SPLINE
SPL {X  -157.404, Y  +360.095, Z    +0.000, E1   +17.695, E3 +134667.595}
SPL {X  -159.413, Y  +375.108, Z    +0.000, E1    +9.284, E3 +134676.684}
SPL {X  -159.978, Y  +386.135, Z    +0.000, E1    +2.544, E3 +134680.245}
SPL {X  -160.000, Y  +393.708, Z    +0.000, E1    -3.216, E3 +134681.999}
SPL {X  -160.000, Y  +400.474, Z    +0.000, E1    -9.529, E3 +134684.045}
SPL {X  -160.000, Y  +409.652, Z    +0.000, E1   -18.026, E3 +134688.182}
SPL {X  -160.000, Y  +437.804, Z    +0.000, E1   -34.779, E3 +134712.975}
SPL {X  -160.000, Y  +463.067, Z    +0.000, E1   -38.672, E3 +134758.675}
SPL {X  -160.000, Y  +469.167, Z    +0.000, E1   -38.717, E3 +134774.781}
SPL {X  -160.000, Y  +476.691, Z    +0.000, E1   -38.728, E3 +134794.712}
SPL {X  -160.000, Y  +483.419, Z    +0.000, E1   -38.692, E3 +134812.613}
SPL {X  -160.000, Y  +489.013, Z    +0.000, E1   -38.683, E3 +134827.451}
SPL {X  -160.000, Y  +494.786, Z    +0.000, E1   -38.693, E3 +134842.761}
SPL {X  -160.000, Y  +500.108, Z    +0.000, E1   -38.668, E3 +134856.913}
SPL {X  -160.000, Y  +504.903, Z    +0.000, E1   -38.673, E3 +134869.634}
SPL {X  -160.000, Y  +510.180, Z    +0.000, E1   -38.675, E3 +134883.638}
SPL {X  -160.000, Y  +515.083, Z    +0.000, E1   -38.662, E3 +134896.658}
SPL {X  -160.000, Y  +520.479, Z    +0.000, E1   -38.692, E3 +134910.932}
SPL {X  -160.000, Y  +525.998, Z    +0.000, E1   -38.666, E3 +134925.611}
SPL {X  -160.000, Y  +531.341, Z    +0.000, E1   -38.684, E3 +134939.755}
SPL {X  -160.000, Y  +537.313, Z    +0.000, E1   -38.686, E3 +134955.595}
SPL {X  -160.000, Y  +543.203, Z    +0.000, E1   -38.679, E3 +134971.220}
SPL {X  -160.000, Y  +551.201, Z    +0.000, E1   -38.768, E3 +134992.281}
SPL {X  -160.000, Y  +561.335, Z    +0.000, E1   -38.777, E3 +135019.152}
SPL {X  -160.000, Y  +568.812, Z    +0.000, E1   -38.671, E3 +135039.155}
SPL {X  -160.000, Y  +574.116, Z    +0.000, E1   -38.680, E3 +135053.225}
SPL {X  -160.000, Y  +582.193, Z    +0.000, E1   -38.759, E3 +135074.529}
SPL {X  -160.000, Y  +591.932, Z    +0.000, E1   -38.763, E3 +135100.354}
SPL {X  -160.000, Y  +601.488, Z    +0.000, E1   -38.747, E3 +135125.729}
SPL {X  -160.000, Y  +609.161, Z    +0.000, E1   -38.685, E3 +135146.181}
SPL {X  -160.000, Y  +614.445, Z    +0.000, E1   -38.661, E3 +135160.230}
SPL {X  -160.000, Y  +621.895, Z    +0.000, E1   -38.769, E3 +135179.818}
SPL {X  -160.000, Y  +631.692, Z    +0.000, E1   -38.748, E3 +135205.871}
SPL {X  -160.000, Y  +639.246, Z    +0.000, E1   -38.671, E3 +135226.047}
SPL {X  -160.000, Y  +644.827, Z    +0.000, E1   -38.662, E3 +135240.882}
SPL {X  -160.000, Y  +650.491, Z    +0.000, E1   -38.673, E3 +135255.869}
SPL {X  -160.000, Y  +656.011, Z    +0.000, E1   -38.669, E3 +135270.522}
SPL {X  -160.000, Y  +661.156, Z    +0.000, E1   -38.659, E3 +135284.197}
SPL {X  -160.000, Y  +666.701, Z    +0.000, E1   -38.683, E3 +135298.858}
SPL {X  -159.961, Y  +675.011, Z    +0.000, E1   -38.755, E3 +135320.844}
SPL {X  -159.451, Y  +684.743, Z    +0.000, E1   -38.666, E3 +135347.198}
SPL {X  -158.386, Y  +694.170, Z    +0.000, E1   -38.484, E3 +135373.316}
SPL {X  -157.286, Y  +700.846, Z    +0.000, E1   -38.194, E3 +135392.284}
SPL {X  -156.328, Y  +705.580, Z    +0.000, E1   -38.037, E3 +135405.820}
SPL {X  -155.162, Y  +710.549, Z    +0.000, E1   -37.822, E3 +135420.224}
SPL {X  -153.914, Y  +715.210, Z    +0.000, E1   -37.596, E3 +135433.873}
SPL {X  -152.686, Y  +719.322, Z    +0.000, E1   -37.361, E3 +135446.045}
SPL {X  -150.251, Y  +726.496, Z    +0.000, E1   -33.848, E3 +135494.541}
ENDSPLINE

SPLINE
SPL {X  -156.089, Y  +706.662, Z    +0.000, E1   -21.279, E3 +135547.194}
SPL {X  -159.059, Y  +688.824, Z    +0.000, E1   -11.551, E3 +135561.155}
SPL {X  -159.959, Y  +675.119, Z    +0.000, E1    -3.373, E3 +135565.983}
SPL {X  -160.000, Y  +666.447, Z    +0.000, E1    +3.005, E3 +135568.018}
SPL {X  -160.000, Y  +658.774, Z    +0.000, E1   +10.317, E3 +135570.276}
SPL {X  -160.000, Y  +647.765, Z    +0.000, E1   +20.359, E3 +135575.642}
SPL {X  -160.000, Y  +622.607, Z    +0.000, E1   +34.692, E3 +135598.509}
SPL {X  -160.000, Y  +593.120, Z    +0.000, E1   +39.775, E3 +135648.039}
SPL {X  -160.000, Y  +586.287, Z    +0.000, E1   +39.762, E3 +135665.506}
SPL {X  -160.000, Y  +577.753, Z    +0.000, E1   +39.844, E3 +135687.147}
SPL {X  -160.000, Y  +567.367, Z    +0.000, E1   +39.853, E3 +135713.642}
SPL {X  -160.000, Y  +559.466, Z    +0.000, E1   +39.761, E3 +135733.923}
SPL {X  -160.000, Y  +552.914, Z    +0.000, E1   +39.787, E3 +135750.590}
SPL {X  -160.000, Y  +546.390, Z    +0.000, E1   +39.760, E3 +135767.304}
SPL {X  -160.000, Y  +540.123, Z    +0.000, E1   +39.770, E3 +135783.283}
SPL {X  -160.000, Y  +533.658, Z    +0.000, E1   +39.771, E3 +135799.782}
SPL {X  -160.000, Y  +527.046, Z    +0.000, E1   +39.771, E3 +135816.658}
SPL {X  -160.000, Y  +521.063, Z    +0.000, E1   +39.756, E3 +135831.942}
SPL {X  -160.000, Y  +515.110, Z    +0.000, E1   +39.770, E3 +135847.115}
SPL {X  -160.000, Y  +508.717, Z    +0.000, E1   +39.766, E3 +135863.433}
SPL {X  -160.000, Y  +502.133, Z    +0.000, E1   +39.780, E3 +135880.199}
ENDSPLINE

SPLINE
SPL {X  -160.000, Y  +512.949, Z    +0.000, E1   +32.050, E3 +135896.457}
ENDSPLINE

SPLINE
SPL {X  -160.000, Y  +507.092, Z    +0.000, E1   +32.805, E3 +135911.085}
SPL {X  -160.000, Y  +499.824, Z    +0.000, E1   +34.003, E3 +135926.827}
SPL {X  -160.000, Y  +491.367, Z    +0.000, E1   +35.449, E3 +135943.568}
SPL {X  -160.000, Y  +483.082, Z    +0.000, E1   +36.782, E3 +135959.406}
SPL {X  -160.000, Y  +474.521, Z    +0.000, E1   +38.037, E3 +135975.494}
SPL {X  -160.000, Y  +465.343, Z    +0.000, E1   +38.802, E3 +135995.653}
SPL {X  -160.000, Y  +457.266, Z    +0.000, E1   +38.756, E3 +136017.107}
SPL {X  -160.000, Y  +448.553, Z    +0.000, E1   +38.823, E3 +136040.058}
SPL {X  -160.000, Y  +439.425, Z    +0.000, E1   +38.797, E3 +136064.229}
SPL {X  -160.000, Y  +430.351, Z    +0.000, E1   +38.810, E3 +136088.244}
SPL {X  -160.000, Y  +421.477, Z    +0.000, E1   +38.792, E3 +136111.747}
SPL {X  -160.000, Y  +412.292, Z    +0.000, E1   +38.825, E3 +136135.975}
SPL {X  -160.000, Y  +403.281, Z    +0.000, E1   +38.797, E3 +136159.855}
SPL {X  -160.000, Y  +394.948, Z    +0.000, E1   +38.796, E3 +136181.896}
SPL {X  -159.971, Y  +385.741, Z    +0.000, E1   +38.831, E3 +136206.218}
SPL {X  -159.525, Y  +376.478, Z    +0.000, E1   +38.739, E3 +136231.209}
SPL {X  -158.721, Y  +368.613, Z    +0.000, E1   +38.561, E3 +136252.932}
SPL {X  -157.505, Y  +360.654, Z    +0.000, E1   +38.390, E3 +136275.205}
SPL {X  -156.229, Y  +354.269, Z    +0.000, E1   +38.076, E3 +136293.555}
SPL {X  -155.202, Y  +349.910, Z    +0.000, E1   +37.893, E3 +136306.129}
SPL {X  -154.128, Y  +345.852, Z    +0.000, E1   +37.701, E3 +136317.953}
SPL {X  -152.890, Y  +341.633, Z    +0.000, E1   +37.487, E3 +136330.385}
SPL {X  -150.284, Y  +333.893, Z    +0.000, E1   +33.433, E3 +136385.195}
ENDSPLINE

SPLINE
SPL {X  -157.404, Y  +360.095, Z    +0.000, E1   +17.695, E3 +136440.320}
SPL {X  -159.413, Y  +375.108, Z    +0.000, E1    +9.284, E3 +136449.409}
SPL {X  -159.978, Y  +386.135, Z    +0.000, E1    +2.544, E3 +136452.970}
SPL {X  -160.000, Y  +393.708, Z    +0.000, E1    -3.216, E3 +136454.724}
SPL {X  -160.000, Y  +400.474, Z    +0.000, E1    -9.529, E3 +136456.771}
SPL {X  -160.000, Y  +409.652, Z    +0.000, E1   -18.026, E3 +136460.907}
SPL {X  -160.000, Y  +437.804, Z    +0.000, E1   -34.779, E3 +136485.700}
SPL {X  -160.000, Y  +463.067, Z    +0.000, E1   -38.672, E3 +136531.400}
SPL {X  -160.000, Y  +469.167, Z    +0.000, E1   -38.717, E3 +136547.506}
SPL {X  -160.000, Y  +476.691, Z    +0.000, E1   -38.728, E3 +136567.438}
SPL {X  -160.000, Y  +483.419, Z    +0.000, E1   -38.692, E3 +136585.338}
SPL {X  -160.000, Y  +489.013, Z    +0.000, E1   -38.683, E3 +136600.177}
SPL {X  -160.000, Y  +494.786, Z    +0.000, E1   -38.693, E3 +136615.487}
SPL {X  -160.000, Y  +500.108, Z    +0.000, E1   -38.668, E3 +136629.638}
SPL {X  -160.000, Y  +504.903, Z    +0.000, E1   -38.673, E3 +136642.359}
SPL {X  -160.000, Y  +510.180, Z    +0.000, E1   -38.675, E3 +136656.363}
SPL {X  -160.000, Y  +515.083, Z    +0.000, E1   -38.662, E3 +136669.383}
SPL {X  -160.000, Y  +520.479, Z    +0.000, E1   -38.692, E3 +136683.658}
SPL {X  -160.000, Y  +525.998, Z    +0.000, E1   -38.666, E3 +136698.336}
SPL {X  -160.000, Y  +531.341, Z    +0.000, E1   -38.684, E3 +136712.480}
SPL {X  -160.000, Y  +537.313, Z    +0.000, E1   -38.686, E3 +136728.320}
SPL {X  -160.000, Y  +543.203, Z    +0.000, E1   -38.679, E3 +136743.945}
SPL {X  -160.000, Y  +551.201, Z    +0.000, E1   -38.768, E3 +136765.007}
SPL {X  -160.000, Y  +561.335, Z    +0.000, E1   -38.777, E3 +136791.877}
SPL {X  -160.000, Y  +568.812, Z    +0.000, E1   -38.671, E3 +136811.880}
SPL {X  -160.000, Y  +574.116, Z    +0.000, E1   -38.680, E3 +136825.951}
SPL {X  -160.000, Y  +582.193, Z    +0.000, E1   -38.759, E3 +136847.254}
SPL {X  -160.000, Y  +591.932, Z    +0.000, E1   -38.763, E3 +136873.079}
SPL {X  -160.000, Y  +601.488, Z    +0.000, E1   -38.747, E3 +136898.454}
SPL {X  -160.000, Y  +609.161, Z    +0.000, E1   -38.685, E3 +136918.906}
SPL {X  -160.000, Y  +614.445, Z    +0.000, E1   -38.661, E3 +136932.955}
SPL {X  -160.000, Y  +621.895, Z    +0.000, E1   -38.769, E3 +136952.543}
SPL {X  -160.000, Y  +631.692, Z    +0.000, E1   -38.748, E3 +136978.597}
SPL {X  -160.000, Y  +639.246, Z    +0.000, E1   -38.671, E3 +136998.772}
SPL {X  -160.000, Y  +644.827, Z    +0.000, E1   -38.662, E3 +137013.607}
SPL {X  -160.000, Y  +650.491, Z    +0.000, E1   -38.673, E3 +137028.595}
SPL {X  -160.000, Y  +656.011, Z    +0.000, E1   -38.669, E3 +137043.248}
SPL {X  -160.000, Y  +661.156, Z    +0.000, E1   -38.659, E3 +137056.923}
SPL {X  -160.000, Y  +666.701, Z    +0.000, E1   -38.683, E3 +137071.583}
SPL {X  -159.961, Y  +675.011, Z    +0.000, E1   -38.755, E3 +137093.569}
SPL {X  -159.451, Y  +684.743, Z    +0.000, E1   -38.666, E3 +137119.923}
SPL {X  -158.386, Y  +694.170, Z    +0.000, E1   -38.484, E3 +137146.041}
SPL {X  -157.286, Y  +700.846, Z    +0.000, E1   -38.194, E3 +137165.009}
SPL {X  -156.328, Y  +705.580, Z    +0.000, E1   -38.037, E3 +137178.545}
SPL {X  -155.162, Y  +710.549, Z    +0.000, E1   -37.822, E3 +137192.949}
SPL {X  -153.914, Y  +715.210, Z    +0.000, E1   -37.596, E3 +137206.598}
SPL {X  -152.686, Y  +719.322, Z    +0.000, E1   -37.361, E3 +137218.771}
SPL {X  -150.251, Y  +726.496, Z    +0.000, E1   -33.848, E3 +137267.266}
ENDSPLINE

SPLINE
SPL {X  -156.089, Y  +706.662, Z    +0.000, E1   -21.279, E3 +137319.920}
SPL {X  -159.059, Y  +688.824, Z    +0.000, E1   -11.551, E3 +137333.880}
SPL {X  -159.959, Y  +675.119, Z    +0.000, E1    -3.373, E3 +137338.708}
SPL {X  -160.000, Y  +666.447, Z    +0.000, E1    +3.005, E3 +137340.743}
SPL {X  -160.000, Y  +658.774, Z    +0.000, E1   +10.317, E3 +137343.002}
SPL {X  -160.000, Y  +647.765, Z    +0.000, E1   +20.359, E3 +137348.367}
SPL {X  -160.000, Y  +622.607, Z    +0.000, E1   +34.692, E3 +137371.234}
SPL {X  -160.000, Y  +596.106, Z    +0.000, E1   +39.718, E3 +137413.234}
SPL {X  -160.000, Y  +592.273, Z    +0.000, E1   +39.746, E3 +137422.972}
SPL {X  -160.000, Y  +586.287, Z    +0.000, E1   +39.762, E3 +137438.231}
SPL {X  -160.000, Y  +577.753, Z    +0.000, E1   +39.844, E3 +137459.873}
SPL {X  -160.000, Y  +567.367, Z    +0.000, E1   +39.853, E3 +137486.367}
SPL {X  -160.000, Y  +559.466, Z    +0.000, E1   +39.761, E3 +137506.648}
SPL {X  -160.000, Y  +552.914, Z    +0.000, E1   +39.787, E3 +137523.316}
SPL {X  -160.000, Y  +546.390, Z    +0.000, E1   +39.760, E3 +137540.029}
SPL {X  -160.000, Y  +540.123, Z    +0.000, E1   +39.770, E3 +137556.009}
SPL {X  -160.000, Y  +533.658, Z    +0.000, E1   +39.771, E3 +137572.507}
SPL {X  -160.000, Y  +527.046, Z    +0.000, E1   +39.771, E3 +137589.383}
SPL {X  -160.000, Y  +521.063, Z    +0.000, E1   +39.756, E3 +137604.667}
SPL {X  -160.000, Y  +515.110, Z    +0.000, E1   +39.770, E3 +137619.840}
SPL {X  -160.000, Y  +508.717, Z    +0.000, E1   +39.766, E3 +137636.158}
SPL {X  -160.000, Y  +502.133, Z    +0.000, E1   +39.780, E3 +137652.925}
ENDSPLINE

SPLINE
SPL {X  -160.000, Y  +512.949, Z    +0.000, E1   +32.050, E3 +137669.182}
ENDSPLINE

SPLINE
SPL {X  -160.000, Y  +507.092, Z    +0.000, E1   +32.805, E3 +137683.810}
SPL {X  -160.000, Y  +499.824, Z    +0.000, E1   +34.003, E3 +137699.552}
SPL {X  -160.000, Y  +491.367, Z    +0.000, E1   +35.449, E3 +137716.293}
SPL {X  -160.000, Y  +483.082, Z    +0.000, E1   +36.782, E3 +137732.132}
SPL {X  -160.000, Y  +474.521, Z    +0.000, E1   +38.037, E3 +137748.220}
SPL {X  -160.000, Y  +465.343, Z    +0.000, E1   +38.802, E3 +137768.378}
SPL {X  -160.000, Y  +457.266, Z    +0.000, E1   +38.756, E3 +137789.832}
SPL {X  -160.000, Y  +448.553, Z    +0.000, E1   +38.823, E3 +137812.783}
SPL {X  -160.000, Y  +439.425, Z    +0.000, E1   +38.797, E3 +137836.954}
SPL {X  -160.000, Y  +430.351, Z    +0.000, E1   +38.810, E3 +137860.969}
SPL {X  -160.000, Y  +421.477, Z    +0.000, E1   +38.792, E3 +137884.472}
SPL {X  -160.000, Y  +412.292, Z    +0.000, E1   +38.825, E3 +137908.700}
SPL {X  -160.000, Y  +403.281, Z    +0.000, E1   +38.797, E3 +137932.580}
SPL {X  -160.000, Y  +394.948, Z    +0.000, E1   +38.796, E3 +137954.621}
SPL {X  -159.971, Y  +385.741, Z    +0.000, E1   +38.831, E3 +137978.943}
SPL {X  -159.525, Y  +376.478, Z    +0.000, E1   +38.739, E3 +138003.934}
SPL {X  -158.721, Y  +368.613, Z    +0.000, E1   +38.561, E3 +138025.657}
SPL {X  -157.505, Y  +360.654, Z    +0.000, E1   +38.390, E3 +138047.930}
SPL {X  -156.229, Y  +354.269, Z    +0.000, E1   +38.076, E3 +138066.280}
SPL {X  -155.202, Y  +349.910, Z    +0.000, E1   +37.893, E3 +138078.854}
SPL {X  -154.128, Y  +345.852, Z    +0.000, E1   +37.701, E3 +138090.678}
SPL {X  -152.890, Y  +341.633, Z    +0.000, E1   +37.487, E3 +138103.110}
SPL {X  -150.284, Y  +333.893, Z    +0.000, E1   +33.433, E3 +138157.921}
ENDSPLINE

SPLINE
SPL {X  -157.404, Y  +360.095, Z    +0.000, E1   +17.695, E3 +138213.045}
SPL {X  -159.413, Y  +375.108, Z    +0.000, E1    +9.284, E3 +138222.134}
SPL {X  -159.978, Y  +386.135, Z    +0.000, E1    +2.544, E3 +138225.695}
SPL {X  -160.000, Y  +393.708, Z    +0.000, E1    -3.216, E3 +138227.449}
SPL {X  -160.000, Y  +400.474, Z    +0.000, E1    -9.529, E3 +138229.496}
SPL {X  -160.000, Y  +409.652, Z    +0.000, E1   -18.026, E3 +138233.632}
SPL {X  -160.000, Y  +437.804, Z    +0.000, E1   -34.779, E3 +138258.425}
SPL {X  -160.000, Y  +463.067, Z    +0.000, E1   -38.672, E3 +138304.125}
SPL {X  -160.000, Y  +469.167, Z    +0.000, E1   -38.717, E3 +138320.231}
SPL {X  -160.000, Y  +476.691, Z    +0.000, E1   -38.728, E3 +138340.163}
SPL {X  -160.000, Y  +483.419, Z    +0.000, E1   -38.692, E3 +138358.063}
SPL {X  -160.000, Y  +489.013, Z    +0.000, E1   -38.683, E3 +138372.902}
SPL {X  -160.000, Y  +494.786, Z    +0.000, E1   -38.693, E3 +138388.212}
SPL {X  -160.000, Y  +500.108, Z    +0.000, E1   -38.668, E3 +138402.363}
SPL {X  -160.000, Y  +504.903, Z    +0.000, E1   -38.673, E3 +138415.084}
SPL {X  -160.000, Y  +510.180, Z    +0.000, E1   -38.675, E3 +138429.089}
SPL {X  -160.000, Y  +515.083, Z    +0.000, E1   -38.662, E3 +138442.108}
SPL {X  -160.000, Y  +520.479, Z    +0.000, E1   -38.692, E3 +138456.383}
SPL {X  -160.000, Y  +525.998, Z    +0.000, E1   -38.666, E3 +138471.061}
SPL {X  -160.000, Y  +531.341, Z    +0.000, E1   -38.684, E3 +138485.205}
SPL {X  -160.000, Y  +537.313, Z    +0.000, E1   -38.686, E3 +138501.045}
SPL {X  -160.000, Y  +543.203, Z    +0.000, E1   -38.679, E3 +138516.671}
SPL {X  -160.000, Y  +551.201, Z    +0.000, E1   -38.768, E3 +138537.732}
SPL {X  -160.000, Y  +561.335, Z    +0.000, E1   -38.777, E3 +138564.602}
SPL {X  -160.000, Y  +568.812, Z    +0.000, E1   -38.671, E3 +138584.605}
SPL {X  -160.000, Y  +574.116, Z    +0.000, E1   -38.680, E3 +138598.676}
SPL {X  -160.000, Y  +582.193, Z    +0.000, E1   -38.759, E3 +138619.979}
SPL {X  -160.000, Y  +591.932, Z    +0.000, E1   -38.763, E3 +138645.804}
SPL {X  -160.000, Y  +601.488, Z    +0.000, E1   -38.747, E3 +138671.179}
SPL {X  -160.000, Y  +609.161, Z    +0.000, E1   -38.685, E3 +138691.631}
SPL {X  -160.000, Y  +614.445, Z    +0.000, E1   -38.661, E3 +138705.680}
SPL {X  -160.000, Y  +621.895, Z    +0.000, E1   -38.769, E3 +138725.269}
SPL {X  -160.000, Y  +631.692, Z    +0.000, E1   -38.748, E3 +138751.322}
SPL {X  -160.000, Y  +639.246, Z    +0.000, E1   -38.671, E3 +138771.498}
SPL {X  -160.000, Y  +644.827, Z    +0.000, E1   -38.662, E3 +138786.332}
SPL {X  -160.000, Y  +650.491, Z    +0.000, E1   -38.673, E3 +138801.320}
SPL {X  -160.000, Y  +656.011, Z    +0.000, E1   -38.669, E3 +138815.973}
SPL {X  -160.000, Y  +661.156, Z    +0.000, E1   -38.659, E3 +138829.648}
SPL {X  -160.000, Y  +666.701, Z    +0.000, E1   -38.683, E3 +138844.308}
SPL {X  -159.961, Y  +675.011, Z    +0.000, E1   -38.755, E3 +138866.295}
SPL {X  -159.451, Y  +684.743, Z    +0.000, E1   -38.666, E3 +138892.648}
SPL {X  -158.386, Y  +694.170, Z    +0.000, E1   -38.484, E3 +138918.767}
SPL {X  -157.286, Y  +700.846, Z    +0.000, E1   -38.194, E3 +138937.734}
SPL {X  -156.328, Y  +705.580, Z    +0.000, E1   -38.037, E3 +138951.270}
SPL {X  -155.162, Y  +710.549, Z    +0.000, E1   -37.822, E3 +138965.674}
SPL {X  -153.914, Y  +715.210, Z    +0.000, E1   -37.596, E3 +138979.324}
SPL {X  -152.686, Y  +719.322, Z    +0.000, E1   -37.361, E3 +138991.496}
SPL {X  -150.251, Y  +726.496, Z    +0.000, E1   -33.848, E3 +139039.992}
ENDSPLINE

SPLINE
SPL {X  -156.089, Y  +706.662, Z    +0.000, E1   -21.279, E3 +139092.645}
SPL {X  -159.059, Y  +688.824, Z    +0.000, E1   -11.551, E3 +139106.605}
SPL {X  -159.959, Y  +675.119, Z    +0.000, E1    -3.373, E3 +139111.433}
SPL {X  -160.000, Y  +666.447, Z    +0.000, E1    +3.005, E3 +139113.468}
SPL {X  -160.000, Y  +658.774, Z    +0.000, E1   +10.317, E3 +139115.727}
SPL {X  -160.000, Y  +647.765, Z    +0.000, E1   +20.359, E3 +139121.092}
SPL {X  -160.000, Y  +622.607, Z    +0.000, E1   +34.692, E3 +139143.959}
SPL {X  -160.000, Y  +596.106, Z    +0.000, E1   +39.718, E3 +139185.959}
SPL {X  -160.000, Y  +592.273, Z    +0.000, E1   +39.746, E3 +139195.697}
SPL {X  -160.000, Y  +586.287, Z    +0.000, E1   +39.762, E3 +139210.956}
SPL {X  -160.000, Y  +577.753, Z    +0.000, E1   +39.844, E3 +139232.598}
SPL {X  -160.000, Y  +567.367, Z    +0.000, E1   +39.853, E3 +139259.092}
SPL {X  -160.000, Y  +559.466, Z    +0.000, E1   +39.761, E3 +139279.373}
SPL {X  -160.000, Y  +552.914, Z    +0.000, E1   +39.787, E3 +139296.041}
SPL {X  -160.000, Y  +546.390, Z    +0.000, E1   +39.760, E3 +139312.755}
SPL {X  -160.000, Y  +540.123, Z    +0.000, E1   +39.770, E3 +139328.734}
SPL {X  -160.000, Y  +533.658, Z    +0.000, E1   +39.771, E3 +139345.232}
SPL {X  -160.000, Y  +527.046, Z    +0.000, E1   +39.771, E3 +139362.108}
SPL {X  -160.000, Y  +521.063, Z    +0.000, E1   +39.756, E3 +139377.393}
SPL {X  -160.000, Y  +515.110, Z    +0.000, E1   +39.770, E3 +139392.565}
SPL {X  -160.000, Y  +508.717, Z    +0.000, E1   +39.766, E3 +139408.884}
SPL {X  -160.000, Y  +502.133, Z    +0.000, E1   +39.780, E3 +139425.650}
ENDSPLINE

SPLINE
SPL {X  -160.000, Y  +512.949, Z    +0.000, E1   +32.050, E3 +139441.907}
ENDSPLINE

SPLINE
SPL {X  -160.000, Y  +507.092, Z    +0.000, E1   +32.805, E3 +139456.536}
SPL {X  -160.000, Y  +499.824, Z    +0.000, E1   +34.003, E3 +139472.277}
SPL {X  -160.000, Y  +491.367, Z    +0.000, E1   +35.449, E3 +139489.018}
SPL {X  -160.000, Y  +483.082, Z    +0.000, E1   +36.782, E3 +139504.857}
SPL {X  -160.000, Y  +474.521, Z    +0.000, E1   +38.037, E3 +139520.945}
SPL {X  -160.000, Y  +465.343, Z    +0.000, E1   +38.802, E3 +139541.104}
SPL {X  -160.000, Y  +457.266, Z    +0.000, E1   +38.756, E3 +139562.557}
SPL {X  -160.000, Y  +448.553, Z    +0.000, E1   +38.823, E3 +139585.508}
SPL {X  -160.000, Y  +439.425, Z    +0.000, E1   +38.797, E3 +139609.679}
SPL {X  -160.000, Y  +430.351, Z    +0.000, E1   +38.810, E3 +139633.694}
SPL {X  -160.000, Y  +421.477, Z    +0.000, E1   +38.792, E3 +139657.198}
SPL {X  -160.000, Y  +412.292, Z    +0.000, E1   +38.825, E3 +139681.425}
SPL {X  -160.000, Y  +403.281, Z    +0.000, E1   +38.797, E3 +139705.305}
SPL {X  -160.000, Y  +394.948, Z    +0.000, E1   +38.796, E3 +139727.347}
SPL {X  -159.971, Y  +385.741, Z    +0.000, E1   +38.831, E3 +139751.668}
SPL {X  -159.525, Y  +376.478, Z    +0.000, E1   +38.739, E3 +139776.659}
SPL {X  -158.721, Y  +368.613, Z    +0.000, E1   +38.561, E3 +139798.382}
SPL {X  -157.505, Y  +360.654, Z    +0.000, E1   +38.390, E3 +139820.655}
SPL {X  -156.229, Y  +354.269, Z    +0.000, E1   +38.076, E3 +139839.005}
SPL {X  -155.202, Y  +349.910, Z    +0.000, E1   +37.893, E3 +139851.580}
SPL {X  -154.128, Y  +345.852, Z    +0.000, E1   +37.701, E3 +139863.404}
SPL {X  -152.890, Y  +341.633, Z    +0.000, E1   +37.487, E3 +139875.836}
SPL {X  -150.284, Y  +333.893, Z    +0.000, E1   +33.433, E3 +139930.646}
ENDSPLINE

SPLINE
SPL {X  -157.404, Y  +360.095, Z    +0.000, E1   +17.695, E3 +139985.771}
SPL {X  -159.413, Y  +375.108, Z    +0.000, E1    +9.284, E3 +139994.860}
SPL {X  -159.978, Y  +386.135, Z    +0.000, E1    +2.544, E3 +139998.421}
SPL {X  -160.000, Y  +393.708, Z    +0.000, E1    -3.216, E3 +140000.175}
SPL {X  -160.000, Y  +400.474, Z    +0.000, E1    -9.529, E3 +140002.221}
SPL {X  -160.000, Y  +409.652, Z    +0.000, E1   -18.026, E3 +140006.358}
SPL {X  -160.000, Y  +437.804, Z    +0.000, E1   -34.779, E3 +140031.150}
SPL {X  -160.000, Y  +463.067, Z    +0.000, E1   -38.672, E3 +140076.850}
SPL {X  -160.000, Y  +469.167, Z    +0.000, E1   -38.717, E3 +140092.956}
SPL {X  -160.000, Y  +476.691, Z    +0.000, E1   -38.728, E3 +140112.888}
SPL {X  -160.000, Y  +483.419, Z    +0.000, E1   -38.692, E3 +140130.788}
SPL {X  -160.000, Y  +489.013, Z    +0.000, E1   -38.683, E3 +140145.627}
SPL {X  -160.000, Y  +494.786, Z    +0.000, E1   -38.693, E3 +140160.937}
SPL {X  -160.000, Y  +500.108, Z    +0.000, E1   -38.668, E3 +140175.089}
SPL {X  -160.000, Y  +504.903, Z    +0.000, E1   -38.673, E3 +140187.810}
SPL {X  -160.000, Y  +510.180, Z    +0.000, E1   -38.675, E3 +140201.814}
SPL {X  -160.000, Y  +515.083, Z    +0.000, E1   -38.662, E3 +140214.834}
SPL {X  -160.000, Y  +520.479, Z    +0.000, E1   -38.692, E3 +140229.108}
SPL {X  -160.000, Y  +525.998, Z    +0.000, E1   -38.666, E3 +140243.786}
SPL {X  -160.000, Y  +531.341, Z    +0.000, E1   -38.684, E3 +140257.930}
SPL {X  -160.000, Y  +537.313, Z    +0.000, E1   -38.686, E3 +140273.770}
SPL {X  -160.000, Y  +543.203, Z    +0.000, E1   -38.679, E3 +140289.396}
SPL {X  -160.000, Y  +551.201, Z    +0.000, E1   -38.768, E3 +140310.457}
SPL {X  -160.000, Y  +561.335, Z    +0.000, E1   -38.777, E3 +140337.327}
SPL {X  -160.000, Y  +568.812, Z    +0.000, E1   -38.671, E3 +140357.331}
SPL {X  -160.000, Y  +574.116, Z    +0.000, E1   -38.680, E3 +140371.401}
SPL {X  -160.000, Y  +582.193, Z    +0.000, E1   -38.759, E3 +140392.705}
SPL {X  -160.000, Y  +591.932, Z    +0.000, E1   -38.763, E3 +140418.530}
SPL {X  -160.000, Y  +601.488, Z    +0.000, E1   -38.747, E3 +140443.905}
SPL {X  -160.000, Y  +609.161, Z    +0.000, E1   -38.685, E3 +140464.357}
SPL {X  -160.000, Y  +614.445, Z    +0.000, E1   -38.661, E3 +140478.406}
SPL {X  -160.000, Y  +621.895, Z    +0.000, E1   -38.769, E3 +140497.994}
SPL {X  -160.000, Y  +631.692, Z    +0.000, E1   -38.748, E3 +140524.047}
SPL {X  -160.000, Y  +639.246, Z    +0.000, E1   -38.671, E3 +140544.223}
SPL {X  -160.000, Y  +644.827, Z    +0.000, E1   -38.662, E3 +140559.058}
SPL {X  -160.000, Y  +650.491, Z    +0.000, E1   -38.673, E3 +140574.045}
SPL {X  -160.000, Y  +656.011, Z    +0.000, E1   -38.669, E3 +140588.698}
SPL {X  -160.000, Y  +661.156, Z    +0.000, E1   -38.659, E3 +140602.373}
SPL {X  -160.000, Y  +666.701, Z    +0.000, E1   -38.683, E3 +140617.033}
SPL {X  -159.961, Y  +675.011, Z    +0.000, E1   -38.755, E3 +140639.020}
SPL {X  -159.451, Y  +684.743, Z    +0.000, E1   -38.666, E3 +140665.373}
SPL {X  -158.386, Y  +694.170, Z    +0.000, E1   -38.484, E3 +140691.492}
SPL {X  -157.286, Y  +700.846, Z    +0.000, E1   -38.194, E3 +140710.460}
SPL {X  -156.328, Y  +705.580, Z    +0.000, E1   -38.037, E3 +140723.996}
SPL {X  -155.162, Y  +710.549, Z    +0.000, E1   -37.822, E3 +140738.399}
SPL {X  -153.914, Y  +715.210, Z    +0.000, E1   -37.596, E3 +140752.049}
SPL {X  -152.686, Y  +719.322, Z    +0.000, E1   -37.361, E3 +140764.221}
SPL {X  -150.251, Y  +726.496, Z    +0.000, E1   -33.848, E3 +140812.717}
ENDSPLINE

SPLINE
SPL {X  -156.089, Y  +706.662, Z    +0.000, E1   -21.279, E3 +140865.370}
SPL {X  -159.059, Y  +688.824, Z    +0.000, E1   -11.551, E3 +140879.331}
SPL {X  -159.959, Y  +675.119, Z    +0.000, E1    -3.373, E3 +140884.159}
SPL {X  -160.000, Y  +666.447, Z    +0.000, E1    +3.005, E3 +140886.194}
SPL {X  -160.000, Y  +658.774, Z    +0.000, E1   +10.317, E3 +140888.452}
SPL {X  -160.000, Y  +647.765, Z    +0.000, E1   +20.359, E3 +140893.817}
SPL {X  -160.000, Y  +622.607, Z    +0.000, E1   +34.692, E3 +140916.685}
SPL {X  -160.000, Y  +593.120, Z    +0.000, E1   +39.775, E3 +140966.215}
SPL {X  -160.000, Y  +586.287, Z    +0.000, E1   +39.762, E3 +140983.681}
SPL {X  -160.000, Y  +577.753, Z    +0.000, E1   +39.844, E3 +141005.323}
SPL {X  -160.000, Y  +567.367, Z    +0.000, E1   +39.853, E3 +141031.817}
SPL {X  -160.000, Y  +559.466, Z    +0.000, E1   +39.761, E3 +141052.099}
SPL {X  -160.000, Y  +552.914, Z    +0.000, E1   +39.787, E3 +141068.766}
SPL {X  -160.000, Y  +546.390, Z    +0.000, E1   +39.760, E3 +141085.480}
SPL {X  -160.000, Y  +540.123, Z    +0.000, E1   +39.770, E3 +141101.459}
SPL {X  -160.000, Y  +533.658, Z    +0.000, E1   +39.771, E3 +141117.958}
SPL {X  -160.000, Y  +527.046, Z    +0.000, E1   +39.771, E3 +141134.833}
SPL {X  -160.000, Y  +521.063, Z    +0.000, E1   +39.756, E3 +141150.118}
SPL {X  -160.000, Y  +515.110, Z    +0.000, E1   +39.770, E3 +141165.290}
SPL {X  -160.000, Y  +508.717, Z    +0.000, E1   +39.766, E3 +141181.609}
SPL {X  -160.000, Y  +502.133, Z    +0.000, E1   +39.780, E3 +141198.375}
ENDSPLINE

SPLINE
SPL {X  -160.000, Y  +512.949, Z    +0.000, E1   +32.050, E3 +141214.633}
ENDSPLINE

SPLINE
SPL {X  -160.000, Y  +507.092, Z    +0.000, E1   +32.805, E3 +141229.261}
SPL {X  -160.000, Y  +499.824, Z    +0.000, E1   +34.003, E3 +141245.003}
SPL {X  -160.000, Y  +491.367, Z    +0.000, E1   +35.449, E3 +141261.743}
SPL {X  -160.000, Y  +483.082, Z    +0.000, E1   +36.782, E3 +141277.582}
SPL {X  -160.000, Y  +474.521, Z    +0.000, E1   +38.037, E3 +141293.670}
SPL {X  -160.000, Y  +465.343, Z    +0.000, E1   +38.802, E3 +141313.829}
SPL {X  -160.000, Y  +457.266, Z    +0.000, E1   +38.756, E3 +141335.283}
SPL {X  -160.000, Y  +448.553, Z    +0.000, E1   +38.823, E3 +141358.234}
SPL {X  -160.000, Y  +439.425, Z    +0.000, E1   +38.797, E3 +141382.405}
SPL {X  -160.000, Y  +430.351, Z    +0.000, E1   +38.810, E3 +141406.419}
SPL {X  -160.000, Y  +421.477, Z    +0.000, E1   +38.792, E3 +141429.923}
SPL {X  -160.000, Y  +412.292, Z    +0.000, E1   +38.825, E3 +141454.150}
SPL {X  -160.000, Y  +403.281, Z    +0.000, E1   +38.797, E3 +141478.030}
SPL {X  -160.000, Y  +394.948, Z    +0.000, E1   +38.796, E3 +141500.072}
SPL {X  -159.971, Y  +385.741, Z    +0.000, E1   +38.831, E3 +141524.393}
SPL {X  -159.525, Y  +376.478, Z    +0.000, E1   +38.739, E3 +141549.384}
SPL {X  -158.721, Y  +368.613, Z    +0.000, E1   +38.561, E3 +141571.107}
SPL {X  -157.505, Y  +360.654, Z    +0.000, E1   +38.390, E3 +141593.381}
SPL {X  -156.229, Y  +354.269, Z    +0.000, E1   +38.076, E3 +141611.730}
SPL {X  -155.202, Y  +349.910, Z    +0.000, E1   +37.893, E3 +141624.305}
SPL {X  -154.128, Y  +345.852, Z    +0.000, E1   +37.701, E3 +141636.129}
SPL {X  -152.890, Y  +341.633, Z    +0.000, E1   +37.487, E3 +141648.561}
SPL {X  -150.284, Y  +333.893, Z    +0.000, E1   +33.433, E3 +141703.371}
ENDSPLINE

SPLINE
SPL {X  -157.404, Y  +360.095, Z    +0.000, E1   +17.695, E3 +141758.496}
SPL {X  -159.413, Y  +375.108, Z    +0.000, E1    +9.284, E3 +141767.585}
SPL {X  -159.978, Y  +386.135, Z    +0.000, E1    +2.544, E3 +141771.146}
SPL {X  -160.000, Y  +393.708, Z    +0.000, E1    -3.216, E3 +141772.900}
SPL {X  -160.000, Y  +400.474, Z    +0.000, E1    -9.529, E3 +141774.946}
SPL {X  -160.000, Y  +409.652, Z    +0.000, E1   -18.026, E3 +141779.083}
SPL {X  -160.000, Y  +437.804, Z    +0.000, E1   -34.779, E3 +141803.876}
SPL {X  -160.000, Y  +463.067, Z    +0.000, E1   -38.672, E3 +141849.576}
SPL {X  -160.000, Y  +469.167, Z    +0.000, E1   -38.717, E3 +141865.682}
SPL {X  -160.000, Y  +476.691, Z    +0.000, E1   -38.728, E3 +141885.613}
SPL {X  -160.000, Y  +483.419, Z    +0.000, E1   -38.692, E3 +141903.514}
SPL {X  -160.000, Y  +489.013, Z    +0.000, E1   -38.683, E3 +141918.352}
SPL {X  -160.000, Y  +494.786, Z    +0.000, E1   -38.693, E3 +141933.662}
SPL {X  -160.000, Y  +500.108, Z    +0.000, E1   -38.668, E3 +141947.814}
SPL {X  -160.000, Y  +504.903, Z    +0.000, E1   -38.673, E3 +141960.535}
SPL {X  -160.000, Y  +510.180, Z    +0.000, E1   -38.675, E3 +141974.539}
SPL {X  -160.000, Y  +515.083, Z    +0.000, E1   -38.662, E3 +141987.559}
SPL {X  -160.000, Y  +520.479, Z    +0.000, E1   -38.692, E3 +142001.833}
SPL {X  -160.000, Y  +525.998, Z    +0.000, E1   -38.666, E3 +142016.512}
SPL {X  -160.000, Y  +531.341, Z    +0.000, E1   -38.684, E3 +142030.656}
SPL {X  -160.000, Y  +537.313, Z    +0.000, E1   -38.686, E3 +142046.495}
SPL {X  -160.000, Y  +543.203, Z    +0.000, E1   -38.679, E3 +142062.121}
SPL {X  -160.000, Y  +551.201, Z    +0.000, E1   -38.768, E3 +142083.182}
SPL {X  -160.000, Y  +561.335, Z    +0.000, E1   -38.777, E3 +142110.053}
SPL {X  -160.000, Y  +568.812, Z    +0.000, E1   -38.671, E3 +142130.056}
SPL {X  -160.000, Y  +574.116, Z    +0.000, E1   -38.680, E3 +142144.126}
SPL {X  -160.000, Y  +582.193, Z    +0.000, E1   -38.759, E3 +142165.430}
SPL {X  -160.000, Y  +591.932, Z    +0.000, E1   -38.763, E3 +142191.255}
SPL {X  -160.000, Y  +601.488, Z    +0.000, E1   -38.747, E3 +142216.630}
SPL {X  -160.000, Y  +609.161, Z    +0.000, E1   -38.685, E3 +142237.082}
SPL {X  -160.000, Y  +614.445, Z    +0.000, E1   -38.661, E3 +142251.131}
SPL {X  -160.000, Y  +621.895, Z    +0.000, E1   -38.769, E3 +142270.719}
SPL {X  -160.000, Y  +631.692, Z    +0.000, E1   -38.748, E3 +142296.772}
SPL {X  -160.000, Y  +639.246, Z    +0.000, E1   -38.671, E3 +142316.948}
SPL {X  -160.000, Y  +644.827, Z    +0.000, E1   -38.662, E3 +142331.783}
SPL {X  -160.000, Y  +650.491, Z    +0.000, E1   -38.673, E3 +142346.770}
SPL {X  -160.000, Y  +656.011, Z    +0.000, E1   -38.669, E3 +142361.423}
SPL {X  -160.000, Y  +661.156, Z    +0.000, E1   -38.659, E3 +142375.098}
SPL {X  -160.000, Y  +666.701, Z    +0.000, E1   -38.683, E3 +142389.759}
SPL {X  -159.961, Y  +675.011, Z    +0.000, E1   -38.755, E3 +142411.745}
SPL {X  -159.451, Y  +684.743, Z    +0.000, E1   -38.666, E3 +142438.099}
SPL {X  -158.386, Y  +694.170, Z    +0.000, E1   -38.484, E3 +142464.217}
SPL {X  -157.286, Y  +700.846, Z    +0.000, E1   -38.194, E3 +142483.185}
SPL {X  -156.328, Y  +705.580, Z    +0.000, E1   -38.037, E3 +142496.721}
SPL {X  -155.162, Y  +710.549, Z    +0.000, E1   -37.822, E3 +142511.125}
SPL {X  -153.914, Y  +715.210, Z    +0.000, E1   -37.596, E3 +142524.774}
SPL {X  -152.686, Y  +719.322, Z    +0.000, E1   -37.361, E3 +142536.946}
SPL {X  -150.251, Y  +726.496, Z    +0.000, E1   -33.848, E3 +142585.442}
ENDSPLINE

SPLINE
SPL {X  -156.089, Y  +706.662, Z    +0.000, E1   -21.279, E3 +142638.095}
SPL {X  -159.059, Y  +688.824, Z    +0.000, E1   -11.551, E3 +142652.056}
SPL {X  -159.959, Y  +675.119, Z    +0.000, E1    -3.373, E3 +142656.884}
SPL {X  -160.000, Y  +666.447, Z    +0.000, E1    +3.005, E3 +142658.919}
SPL {X  -160.000, Y  +658.774, Z    +0.000, E1   +10.317, E3 +142661.177}
SPL {X  -160.000, Y  +647.765, Z    +0.000, E1   +20.359, E3 +142666.542}
SPL {X  -160.000, Y  +622.607, Z    +0.000, E1   +34.692, E3 +142689.410}
SPL {X  -160.000, Y  +596.106, Z    +0.000, E1   +39.718, E3 +142731.410}
SPL {X  -160.000, Y  +592.273, Z    +0.000, E1   +39.746, E3 +142741.147}
SPL {X  -160.000, Y  +586.287, Z    +0.000, E1   +39.762, E3 +142756.407}
SPL {X  -160.000, Y  +577.753, Z    +0.000, E1   +39.844, E3 +142778.048}
SPL {X  -160.000, Y  +567.367, Z    +0.000, E1   +39.853, E3 +142804.542}
SPL {X  -160.000, Y  +559.466, Z    +0.000, E1   +39.761, E3 +142824.824}
SPL {X  -160.000, Y  +552.914, Z    +0.000, E1   +39.787, E3 +142841.491}
SPL {X  -160.000, Y  +546.390, Z    +0.000, E1   +39.760, E3 +142858.205}
SPL {X  -160.000, Y  +540.123, Z    +0.000, E1   +39.770, E3 +142874.184}
SPL {X  -160.000, Y  +533.658, Z    +0.000, E1   +39.771, E3 +142890.683}
SPL {X  -160.000, Y  +527.046, Z    +0.000, E1   +39.771, E3 +142907.559}
SPL {X  -160.000, Y  +521.063, Z    +0.000, E1   +39.756, E3 +142922.843}
SPL {X  -160.000, Y  +515.110, Z    +0.000, E1   +39.770, E3 +142938.016}
SPL {X  -160.000, Y  +508.717, Z    +0.000, E1   +39.766, E3 +142954.334}
SPL {X  -160.000, Y  +502.133, Z    +0.000, E1   +39.780, E3 +142971.100}
ENDSPLINE

SPLINE
SPL {X  -160.000, Y  +512.949, Z    +0.000, E1   +32.050, E3 +142987.358}
ENDSPLINE

SPLINE
SPL {X  -160.000, Y  +507.092, Z    +0.000, E1   +32.805, E3 +143001.986}
SPL {X  -160.000, Y  +499.824, Z    +0.000, E1   +34.003, E3 +143017.728}
SPL {X  -160.000, Y  +491.367, Z    +0.000, E1   +35.449, E3 +143034.469}
SPL {X  -160.000, Y  +483.082, Z    +0.000, E1   +36.782, E3 +143050.307}
SPL {X  -160.000, Y  +474.521, Z    +0.000, E1   +38.037, E3 +143066.395}
SPL {X  -160.000, Y  +465.343, Z    +0.000, E1   +38.802, E3 +143086.554}
SPL {X  -160.000, Y  +457.266, Z    +0.000, E1   +38.756, E3 +143108.008}
SPL {X  -160.000, Y  +448.553, Z    +0.000, E1   +38.823, E3 +143130.959}
SPL {X  -160.000, Y  +439.425, Z    +0.000, E1   +38.797, E3 +143155.130}
SPL {X  -160.000, Y  +430.351, Z    +0.000, E1   +38.810, E3 +143179.145}
SPL {X  -160.000, Y  +421.477, Z    +0.000, E1   +38.792, E3 +143202.648}
SPL {X  -160.000, Y  +412.292, Z    +0.000, E1   +38.825, E3 +143226.876}
SPL {X  -160.000, Y  +403.281, Z    +0.000, E1   +38.797, E3 +143250.756}
SPL {X  -160.000, Y  +394.948, Z    +0.000, E1   +38.796, E3 +143272.797}
SPL {X  -159.971, Y  +385.741, Z    +0.000, E1   +38.831, E3 +143297.119}
SPL {X  -159.525, Y  +376.478, Z    +0.000, E1   +38.739, E3 +143322.110}
SPL {X  -158.721, Y  +368.613, Z    +0.000, E1   +38.561, E3 +143343.833}
SPL {X  -157.505, Y  +360.654, Z    +0.000, E1   +38.390, E3 +143366.106}
SPL {X  -156.229, Y  +354.269, Z    +0.000, E1   +38.076, E3 +143384.456}
SPL {X  -155.202, Y  +349.910, Z    +0.000, E1   +37.893, E3 +143397.030}
SPL {X  -154.128, Y  +345.852, Z    +0.000, E1   +37.701, E3 +143408.854}
SPL {X  -152.890, Y  +341.633, Z    +0.000, E1   +37.487, E3 +143421.286}
SPL {X  -150.284, Y  +333.893, Z    +0.000, E1   +33.433, E3 +143476.096}
ENDSPLINE

SPLINE
SPL {X  -157.404, Y  +360.095, Z    +0.000, E1   +17.695, E3 +143531.221}
SPL {X  -159.413, Y  +375.108, Z    +0.000, E1    +9.284, E3 +143540.310}
SPL {X  -159.978, Y  +386.135, Z    +0.000, E1    +2.544, E3 +143543.871}
SPL {X  -160.000, Y  +393.708, Z    +0.000, E1    -3.216, E3 +143545.625}
SPL {X  -160.000, Y  +400.474, Z    +0.000, E1    -9.529, E3 +143547.671}
SPL {X  -160.000, Y  +409.652, Z    +0.000, E1   -18.026, E3 +143551.808}
SPL {X  -160.000, Y  +437.804, Z    +0.000, E1   -34.779, E3 +143576.601}
SPL {X  -160.000, Y  +463.067, Z    +0.000, E1   -38.672, E3 +143622.301}
SPL {X  -160.000, Y  +469.167, Z    +0.000, E1   -38.717, E3 +143638.407}
SPL {X  -160.000, Y  +476.691, Z    +0.000, E1   -38.728, E3 +143658.339}
SPL {X  -160.000, Y  +483.419, Z    +0.000, E1   -38.692, E3 +143676.239}
SPL {X  -160.000, Y  +489.013, Z    +0.000, E1   -38.683, E3 +143691.078}
SPL {X  -160.000, Y  +494.786, Z    +0.000, E1   -38.693, E3 +143706.388}
SPL {X  -160.000, Y  +500.108, Z    +0.000, E1   -38.668, E3 +143720.539}
SPL {X  -160.000, Y  +504.903, Z    +0.000, E1   -38.673, E3 +143733.260}
SPL {X  -160.000, Y  +510.180, Z    +0.000, E1   -38.675, E3 +143747.264}
SPL {X  -160.000, Y  +515.083, Z    +0.000, E1   -38.662, E3 +143760.284}
SPL {X  -160.000, Y  +520.479, Z    +0.000, E1   -38.692, E3 +143774.559}
SPL {X  -160.000, Y  +525.998, Z    +0.000, E1   -38.666, E3 +143789.237}
SPL {X  -160.000, Y  +531.341, Z    +0.000, E1   -38.684, E3 +143803.381}
SPL {X  -160.000, Y  +537.313, Z    +0.000, E1   -38.686, E3 +143819.221}
SPL {X  -160.000, Y  +543.203, Z    +0.000, E1   -38.679, E3 +143834.846}
SPL {X  -160.000, Y  +551.201, Z    +0.000, E1   -38.768, E3 +143855.908}
SPL {X  -160.000, Y  +561.335, Z    +0.000, E1   -38.777, E3 +143882.778}
SPL {X  -160.000, Y  +568.812, Z    +0.000, E1   -38.671, E3 +143902.781}
SPL {X  -160.000, Y  +574.116, Z    +0.000, E1   -38.680, E3 +143916.852}
SPL {X  -160.000, Y  +582.193, Z    +0.000, E1   -38.759, E3 +143938.155}
SPL {X  -160.000, Y  +591.932, Z    +0.000, E1   -38.763, E3 +143963.980}
SPL {X  -160.000, Y  +601.488, Z    +0.000, E1   -38.747, E3 +143989.355}
SPL {X  -160.000, Y  +609.161, Z    +0.000, E1   -38.685, E3 +144009.807}
SPL {X  -160.000, Y  +614.445, Z    +0.000, E1   -38.661, E3 +144023.856}
SPL {X  -160.000, Y  +621.895, Z    +0.000, E1   -38.769, E3 +144043.444}
SPL {X  -160.000, Y  +631.692, Z    +0.000, E1   -38.748, E3 +144069.498}
SPL {X  -160.000, Y  +639.246, Z    +0.000, E1   -38.671, E3 +144089.673}
SPL {X  -160.000, Y  +644.827, Z    +0.000, E1   -38.662, E3 +144104.508}
SPL {X  -160.000, Y  +650.491, Z    +0.000, E1   -38.673, E3 +144119.495}
SPL {X  -160.000, Y  +656.011, Z    +0.000, E1   -38.669, E3 +144134.148}
SPL {X  -160.000, Y  +661.156, Z    +0.000, E1   -38.659, E3 +144147.824}
SPL {X  -160.000, Y  +666.701, Z    +0.000, E1   -38.683, E3 +144162.484}
SPL {X  -159.961, Y  +675.011, Z    +0.000, E1   -38.755, E3 +144184.470}
SPL {X  -159.451, Y  +684.743, Z    +0.000, E1   -38.666, E3 +144210.824}
SPL {X  -158.386, Y  +694.170, Z    +0.000, E1   -38.484, E3 +144236.942}
SPL {X  -157.286, Y  +700.846, Z    +0.000, E1   -38.194, E3 +144255.910}
SPL {X  -156.328, Y  +705.580, Z    +0.000, E1   -38.037, E3 +144269.446}
SPL {X  -155.162, Y  +710.549, Z    +0.000, E1   -37.822, E3 +144283.850}
SPL {X  -153.914, Y  +715.210, Z    +0.000, E1   -37.596, E3 +144297.499}
SPL {X  -152.686, Y  +719.322, Z    +0.000, E1   -37.361, E3 +144309.672}
SPL {X  -150.251, Y  +726.496, Z    +0.000, E1   -33.848, E3 +144358.167}
ENDSPLINE

SPLINE
SPL {X  -156.089, Y  +706.662, Z    +0.000, E1   -21.279, E3 +144410.821}
SPL {X  -159.059, Y  +688.824, Z    +0.000, E1   -11.551, E3 +144424.781}
SPL {X  -159.959, Y  +675.119, Z    +0.000, E1    -3.373, E3 +144429.609}
SPL {X  -160.000, Y  +666.447, Z    +0.000, E1    +3.005, E3 +144431.644}
SPL {X  -160.000, Y  +658.774, Z    +0.000, E1   +10.317, E3 +144433.903}
SPL {X  -160.000, Y  +647.765, Z    +0.000, E1   +20.359, E3 +144439.268}
SPL {X  -160.000, Y  +622.607, Z    +0.000, E1   +34.692, E3 +144462.135}
SPL {X  -160.000, Y  +593.120, Z    +0.000, E1   +39.775, E3 +144511.665}
SPL {X  -160.000, Y  +586.287, Z    +0.000, E1   +39.762, E3 +144529.132}
SPL {X  -160.000, Y  +577.753, Z    +0.000, E1   +39.844, E3 +144550.774}
SPL {X  -160.000, Y  +567.367, Z    +0.000, E1   +39.853, E3 +144577.268}
SPL {X  -160.000, Y  +559.466, Z    +0.000, E1   +39.761, E3 +144597.549}
SPL {X  -160.000, Y  +552.914, Z    +0.000, E1   +39.787, E3 +144614.217}
SPL {X  -160.000, Y  +546.390, Z    +0.000, E1   +39.760, E3 +144630.930}
SPL {X  -160.000, Y  +540.123, Z    +0.000, E1   +39.770, E3 +144646.910}
SPL {X  -160.000, Y  +533.658, Z    +0.000, E1   +39.771, E3 +144663.408}
SPL {X  -160.000, Y  +527.046, Z    +0.000, E1   +39.771, E3 +144680.284}
SPL {X  -160.000, Y  +521.063, Z    +0.000, E1   +39.756, E3 +144695.568}
SPL {X  -160.000, Y  +515.110, Z    +0.000, E1   +39.770, E3 +144710.741}
SPL {X  -160.000, Y  +508.717, Z    +0.000, E1   +39.766, E3 +144727.059}
SPL {X  -160.000, Y  +502.133, Z    +0.000, E1   +39.780, E3 +144743.826}
ENDSPLINE

SPLINE
SPL {X  -160.000, Y  +512.949, Z    +0.000, E1   +32.050, E3 +144760.083}
ENDSPLINE

SPLINE
SPL {X  -160.000, Y  +507.092, Z    +0.000, E1   +32.805, E3 +144774.711}
SPL {X  -160.000, Y  +499.824, Z    +0.000, E1   +34.003, E3 +144790.453}
SPL {X  -160.000, Y  +491.367, Z    +0.000, E1   +35.449, E3 +144807.194}
SPL {X  -160.000, Y  +483.082, Z    +0.000, E1   +36.782, E3 +144823.033}
SPL {X  -160.000, Y  +474.521, Z    +0.000, E1   +38.037, E3 +144839.121}
SPL {X  -160.000, Y  +465.343, Z    +0.000, E1   +38.802, E3 +144859.279}
SPL {X  -160.000, Y  +457.266, Z    +0.000, E1   +38.756, E3 +144880.733}
SPL {X  -160.000, Y  +448.553, Z    +0.000, E1   +38.823, E3 +144903.684}
SPL {X  -160.000, Y  +439.425, Z    +0.000, E1   +38.797, E3 +144927.855}
SPL {X  -160.000, Y  +430.351, Z    +0.000, E1   +38.810, E3 +144951.870}
SPL {X  -160.000, Y  +421.477, Z    +0.000, E1   +38.792, E3 +144975.373}
SPL {X  -160.000, Y  +412.292, Z    +0.000, E1   +38.825, E3 +144999.601}
SPL {X  -160.000, Y  +403.281, Z    +0.000, E1   +38.797, E3 +145023.481}
SPL {X  -160.000, Y  +394.948, Z    +0.000, E1   +38.796, E3 +145045.522}
SPL {X  -159.971, Y  +385.741, Z    +0.000, E1   +38.831, E3 +145069.844}
SPL {X  -159.525, Y  +376.478, Z    +0.000, E1   +38.739, E3 +145094.835}
SPL {X  -158.721, Y  +368.613, Z    +0.000, E1   +38.561, E3 +145116.558}
SPL {X  -157.505, Y  +360.654, Z    +0.000, E1   +38.390, E3 +145138.831}
SPL {X  -156.229, Y  +354.269, Z    +0.000, E1   +38.076, E3 +145157.181}
SPL {X  -155.202, Y  +349.910, Z    +0.000, E1   +37.893, E3 +145169.755}
SPL {X  -154.128, Y  +345.852, Z    +0.000, E1   +37.701, E3 +145181.579}
SPL {X  -152.890, Y  +341.633, Z    +0.000, E1   +37.487, E3 +145194.011}
SPL {X  -150.284, Y  +333.893, Z    +0.000, E1   +33.433, E3 +145248.822}
ENDSPLINE

SPLINE
SPL {X  -157.404, Y  +360.095, Z    +0.000, E1   +17.695, E3 +145303.946}
SPL {X  -159.413, Y  +375.108, Z    +0.000, E1    +9.284, E3 +145313.035}
SPL {X  -159.978, Y  +386.135, Z    +0.000, E1    +2.544, E3 +145316.596}
SPL {X  -160.000, Y  +393.708, Z    +0.000, E1    -3.216, E3 +145318.350}
SPL {X  -160.000, Y  +400.474, Z    +0.000, E1    -9.529, E3 +145320.397}
SPL {X  -160.000, Y  +409.652, Z    +0.000, E1   -18.026, E3 +145324.533}
SPL {X  -160.000, Y  +437.804, Z    +0.000, E1   -34.779, E3 +145349.326}
SPL {X  -160.000, Y  +463.067, Z    +0.000, E1   -38.672, E3 +145395.026}
SPL {X  -160.000, Y  +469.167, Z    +0.000, E1   -38.717, E3 +145411.132}
SPL {X  -160.000, Y  +476.691, Z    +0.000, E1   -38.728, E3 +145431.064}
SPL {X  -160.000, Y  +483.419, Z    +0.000, E1   -38.692, E3 +145448.964}
SPL {X  -160.000, Y  +489.013, Z    +0.000, E1   -38.683, E3 +145463.803}
SPL {X  -160.000, Y  +494.786, Z    +0.000, E1   -38.693, E3 +145479.113}
SPL {X  -160.000, Y  +500.108, Z    +0.000, E1   -38.668, E3 +145493.264}
SPL {X  -160.000, Y  +504.903, Z    +0.000, E1   -38.673, E3 +145505.985}
SPL {X  -160.000, Y  +510.180, Z    +0.000, E1   -38.675, E3 +145519.990}
SPL {X  -160.000, Y  +515.083, Z    +0.000, E1   -38.662, E3 +145533.009}
SPL {X  -160.000, Y  +520.479, Z    +0.000, E1   -38.692, E3 +145547.284}
SPL {X  -160.000, Y  +525.998, Z    +0.000, E1   -38.666, E3 +145561.962}
SPL {X  -160.000, Y  +531.341, Z    +0.000, E1   -38.684, E3 +145576.106}
SPL {X  -160.000, Y  +537.313, Z    +0.000, E1   -38.686, E3 +145591.946}
SPL {X  -160.000, Y  +543.203, Z    +0.000, E1   -38.679, E3 +145607.572}
SPL {X  -160.000, Y  +551.201, Z    +0.000, E1   -38.768, E3 +145628.633}
SPL {X  -160.000, Y  +561.335, Z    +0.000, E1   -38.777, E3 +145655.503}
SPL {X  -160.000, Y  +568.812, Z    +0.000, E1   -38.671, E3 +145675.506}
SPL {X  -160.000, Y  +574.116, Z    +0.000, E1   -38.680, E3 +145689.577}
SPL {X  -160.000, Y  +582.193, Z    +0.000, E1   -38.759, E3 +145710.880}
SPL {X  -160.000, Y  +591.932, Z    +0.000, E1   -38.763, E3 +145736.705}
SPL {X  -160.000, Y  +601.488, Z    +0.000, E1   -38.747, E3 +145762.080}
SPL {X  -160.000, Y  +609.161, Z    +0.000, E1   -38.685, E3 +145782.532}
SPL {X  -160.000, Y  +614.445, Z    +0.000, E1   -38.661, E3 +145796.581}
SPL {X  -160.000, Y  +621.895, Z    +0.000, E1   -38.769, E3 +145816.170}
SPL {X  -160.000, Y  +631.692, Z    +0.000, E1   -38.748, E3 +145842.223}
SPL {X  -160.000, Y  +639.246, Z    +0.000, E1   -38.671, E3 +145862.399}
SPL {X  -160.000, Y  +644.827, Z    +0.000, E1   -38.662, E3 +145877.233}
SPL {X  -160.000, Y  +650.491, Z    +0.000, E1   -38.673, E3 +145892.221}
SPL {X  -160.000, Y  +656.011, Z    +0.000, E1   -38.669, E3 +145906.874}
SPL {X  -160.000, Y  +661.156, Z    +0.000, E1   -38.659, E3 +145920.549}
SPL {X  -160.000, Y  +666.701, Z    +0.000, E1   -38.683, E3 +145935.209}
SPL {X  -159.961, Y  +675.011, Z    +0.000, E1   -38.755, E3 +145957.195}
SPL {X  -159.451, Y  +684.743, Z    +0.000, E1   -38.666, E3 +145983.549}
SPL {X  -158.386, Y  +694.170, Z    +0.000, E1   -38.484, E3 +146009.668}
SPL {X  -157.286, Y  +700.846, Z    +0.000, E1   -38.194, E3 +146028.635}
SPL {X  -156.328, Y  +705.580, Z    +0.000, E1   -38.037, E3 +146042.171}
SPL {X  -155.162, Y  +710.549, Z    +0.000, E1   -37.822, E3 +146056.575}
SPL {X  -153.914, Y  +715.210, Z    +0.000, E1   -37.596, E3 +146070.225}
SPL {X  -152.686, Y  +719.322, Z    +0.000, E1   -37.361, E3 +146082.397}
SPL {X  -150.251, Y  +726.496, Z    +0.000, E1   -33.848, E3 +146130.893}
ENDSPLINE

SPLINE
SPL {X  -156.089, Y  +706.662, Z    +0.000, E1   -21.279, E3 +146183.546}
SPL {X  -159.059, Y  +688.824, Z    +0.000, E1   -11.551, E3 +146197.506}
SPL {X  -159.959, Y  +675.119, Z    +0.000, E1    -3.373, E3 +146202.334}
SPL {X  -160.000, Y  +666.447, Z    +0.000, E1    +3.005, E3 +146204.369}
SPL {X  -160.000, Y  +658.774, Z    +0.000, E1   +10.317, E3 +146206.628}
SPL {X  -160.000, Y  +647.765, Z    +0.000, E1   +20.359, E3 +146211.993}
SPL {X  -160.000, Y  +622.607, Z    +0.000, E1   +34.692, E3 +146234.860}
SPL {X  -160.000, Y  +596.106, Z    +0.000, E1   +39.718, E3 +146276.860}
SPL {X  -160.000, Y  +592.273, Z    +0.000, E1   +39.746, E3 +146286.598}
SPL {X  -160.000, Y  +586.287, Z    +0.000, E1   +39.762, E3 +146301.857}
SPL {X  -160.000, Y  +577.753, Z    +0.000, E1   +39.844, E3 +146323.499}
SPL {X  -160.000, Y  +567.367, Z    +0.000, E1   +39.853, E3 +146349.993}
SPL {X  -160.000, Y  +559.466, Z    +0.000, E1   +39.761, E3 +146370.274}
SPL {X  -160.000, Y  +552.914, Z    +0.000, E1   +39.787, E3 +146386.942}
SPL {X  -160.000, Y  +546.390, Z    +0.000, E1   +39.760, E3 +146403.655}
SPL {X  -160.000, Y  +540.123, Z    +0.000, E1   +39.770, E3 +146419.635}
SPL {X  -160.000, Y  +533.658, Z    +0.000, E1   +39.771, E3 +146436.133}
SPL {X  -160.000, Y  +527.046, Z    +0.000, E1   +39.771, E3 +146453.009}
SPL {X  -160.000, Y  +521.063, Z    +0.000, E1   +39.756, E3 +146468.294}
SPL {X  -160.000, Y  +515.110, Z    +0.000, E1   +39.770, E3 +146483.466}
SPL {X  -160.000, Y  +508.717, Z    +0.000, E1   +39.766, E3 +146499.785}
SPL {X  -160.000, Y  +502.133, Z    +0.000, E1   +39.780, E3 +146516.551}
ENDSPLINE

SPLINE
SPL {X  -160.000, Y  +512.949, Z    +0.000, E1   +32.050, E3 +146532.808}
ENDSPLINE

SPLINE
SPL {X  -160.000, Y  +507.092, Z    +0.000, E1   +32.805, E3 +146547.437}
SPL {X  -160.000, Y  +499.824, Z    +0.000, E1   +34.003, E3 +146563.178}
SPL {X  -160.000, Y  +491.367, Z    +0.000, E1   +35.449, E3 +146579.919}
SPL {X  -160.000, Y  +483.082, Z    +0.000, E1   +36.782, E3 +146595.758}
SPL {X  -160.000, Y  +474.521, Z    +0.000, E1   +38.037, E3 +146611.846}
ENDSPLINE

SPLINE
SPL {X  -160.000, Y  +484.185, Z    +0.000, E1   +31.002, E3 +146626.419}
SPL {X  -160.000, Y  +479.156, Z    +0.000, E1   +31.035, E3 +146644.137}
SPL {X  -160.000, Y  +474.045, Z    +0.000, E1   +31.015, E3 +146662.229}
SPL {X  -160.000, Y  +468.999, Z    +0.000, E1   +31.021, E3 +146680.054}
SPL {X  -160.000, Y  +464.107, Z    +0.000, E1   +31.012, E3 +146697.354}
SPL {X  -160.000, Y  +459.262, Z    +0.000, E1   +31.016, E3 +146714.461}
SPL {X  -160.000, Y  +454.119, Z    +0.000, E1   +31.026, E3 +146732.610}
SPL {X  -160.000, Y  +448.874, Z    +0.000, E1   +31.019, E3 +146751.166}
SPL {X  -160.000, Y  +443.892, Z    +0.000, E1   +31.019, E3 +146768.754}
SPL {X  -160.000, Y  +438.782, Z    +0.000, E1   +31.022, E3 +146786.829}
SPL {X  -160.000, Y  +433.722, Z    +0.000, E1   +31.007, E3 +146804.772}
SPL {X  -160.000, Y  +428.980, Z    +0.000, E1   +31.004, E3 +146821.530}
SPL {X  -160.000, Y  +424.339, Z    +0.000, E1   +31.006, E3 +146837.904}
SPL {X  -160.000, Y  +419.231, Z    +0.000, E1   +31.030, E3 +146855.897}
SPL {X  -160.000, Y  +414.179, Z    +0.000, E1   +31.008, E3 +146873.795}
SPL {X  -160.000, Y  +409.416, Z    +0.000, E1   +31.023, E3 +146890.578}
SPL {X  -160.000, Y  +403.994, Z    +0.000, E1   +31.033, E3 +146909.733}
SPL {X  -160.000, Y  +399.052, Z    +0.000, E1   +31.010, E3 +146927.201}
SPL {X  -160.000, Y  +394.012, Z    +0.000, E1   +31.036, E3 +146944.990}
SPL {X  -159.999, Y  +388.376, Z    +0.000, E1   +31.028, E3 +146964.920}
SPL {X  -159.897, Y  +383.070, Z    +0.000, E1   +31.010, E3 +146983.758}
SPL {X  -159.656, Y  +378.313, Z    +0.000, E1   +30.961, E3 +147000.850}
SPL {X  -159.237, Y  +373.190, Z    +0.000, E1   +30.917, E3 +147019.350}
SPL {X  -158.628, Y  +367.891, Z    +0.000, E1   +30.812, E3 +147038.736}
SPL {X  -157.915, Y  +363.053, Z    +0.000, E1   +30.689, E3 +147056.603}
SPL {X  -157.216, Y  +359.084, Z    +0.000, E1   +30.550, E3 +147071.406}
SPL {X  -156.248, Y  +354.355, Z    +0.000, E1   +30.460, E3 +147089.018}
SPL {X  -155.629, Y  +351.657, Z    +0.000, E1   +25.972, E3 +147135.446}
ENDSPLINE

SPLINE
SPL {X  -156.240, Y  +354.319, Z    +0.000, E1   +23.538, E3 +147148.054}
SPL {X  -159.137, Y  +372.201, Z    +0.000, E1   +12.017, E3 +147177.891}
SPL {X  -159.858, Y  +382.069, Z    +0.000, E1    +5.945, E3 +147184.409}
SPL {X  -160.000, Y  +389.339, Z    +0.000, E1    +1.101, E3 +147187.571}
SPL {X  -160.000, Y  +395.749, Z    +0.000, E1    -3.722, E3 +147190.176}
SPL {X  -160.000, Y  +403.128, Z    +0.000, E1    -9.899, E3 +147193.480}
SPL {X  -160.000, Y  +411.609, Z    +0.000, E1   -16.851, E3 +147198.801}
SPL {X  -160.000, Y  +429.715, Z    +0.000, E1   -27.376, E3 +147218.165}
SPL {X  -160.000, Y  +449.791, Z    +0.000, E1   -32.145, E3 +147259.402}
SPL {X  -160.000, Y  +454.903, Z    +0.000, E1   -32.134, E3 +147276.706}
SPL {X  -160.000, Y  +460.041, Z    +0.000, E1   -32.144, E3 +147294.060}
SPL {X  -160.000, Y  +465.466, Z    +0.000, E1   -32.152, E3 +147312.378}
SPL {X  -160.000, Y  +471.112, Z    +0.000, E1   -32.154, E3 +147331.466}
SPL {X  -160.000, Y  +476.735, Z    +0.000, E1   -32.156, E3 +147350.457}
SPL {X  -160.000, Y  +482.675, Z    +0.000, E1   -32.169, E3 +147370.506}
SPL {X  -160.000, Y  +488.008, Z    +0.000, E1   -32.144, E3 +147388.552}
SPL {X  -160.000, Y  +493.245, Z    +0.000, E1   -32.159, E3 +147406.260}
SPL {X  -160.000, Y  +498.210, Z    +0.000, E1   -32.128, E3 +147423.095}
SPL {X  -160.000, Y  +503.407, Z    +0.000, E1   -32.165, E3 +147440.599}
SPL {X  -160.000, Y  +509.142, Z    +0.000, E1   -32.157, E3 +147459.994}
SPL {X  -160.000, Y  +514.696, Z    +0.000, E1   -32.156, E3 +147478.775}
SPL {X  -160.000, Y  +520.339, Z    +0.000, E1   -32.159, E3 +147497.847}
SPL {X  -160.000, Y  +525.825, Z    +0.000, E1   -32.148, E3 +147516.410}
SPL {X  -160.000, Y  +530.379, Z    +0.000, E1   -32.130, E3 +147531.839}
SPL {X  -160.000, Y  +535.020, Z    +0.000, E1   -32.146, E3 +147547.485}
SPL {X  -160.000, Y  +540.303, Z    +0.000, E1   -32.158, E3 +147565.310}
SPL {X  -160.000, Y  +545.740, Z    +0.000, E1   -32.155, E3 +147583.703}
SPL {X  -160.000, Y  +550.807, Z    +0.000, E1   -32.147, E3 +147600.825}
SPL {X  -160.000, Y  +555.841, Z    +0.000, E1   -32.148, E3 +147617.865}
SPL {X  -160.000, Y  +561.018, Z    +0.000, E1   -32.143, E3 +147635.393}
SPL {X  -160.000, Y  +566.466, Z    +0.000, E1   -32.153, E3 +147653.811}
SPL {X  -160.000, Y  +571.733, Z    +0.000, E1   -32.135, E3 +147671.648}
SPL {X  -160.000, Y  +576.943, Z    +0.000, E1   -32.148, E3 +147689.245}
SPL {X  -160.000, Y  +582.183, Z    +0.000, E1   -32.140, E3 +147706.970}
SPL {X  -160.000, Y  +587.036, Z    +0.000, E1   -32.141, E3 +147723.341}
SPL {X  -160.000, Y  +591.785, Z    +0.000, E1   -32.144, E3 +147739.364}
SPL {X  -160.000, Y  +596.962, Z    +0.000, E1   -32.161, E3 +147756.851}
SPL {X  -160.000, Y  +601.800, Z    +0.000, E1   -32.134, E3 +147773.248}
SPL {X  -160.000, Y  +606.611, Z    +0.000, E1   -32.156, E3 +147789.462}
SPL {X  -160.000, Y  +611.219, Z    +0.000, E1   -32.131, E3 +147805.076}
SPL {X  -160.000, Y  +616.331, Z    +0.000, E1   -32.174, E3 +147822.274}
SPL {X  -160.000, Y  +621.751, Z    +0.000, E1   -32.150, E3 +147840.616}
SPL {X  -160.000, Y  +626.312, Z    +0.000, E1   -32.145, E3 +147856.022}
SPL {X  -160.000, Y  +630.971, Z    +0.000, E1   -32.155, E3 +147871.750}
SPL {X  -160.000, Y  +635.550, Z    +0.000, E1   -32.137, E3 +147887.276}
SPL {X  -160.000, Y  +640.419, Z    +0.000, E1   -32.158, E3 +147903.714}
SPL {X  -160.000, Y  +645.749, Z    +0.000, E1   -32.151, E3 +147921.740}
SPL {X  -160.000, Y  +650.662, Z    +0.000, E1   -32.150, E3 +147938.311}
SPL {X  -160.000, Y  +655.372, Z    +0.000, E1   -32.145, E3 +147954.258}
SPL {X  -160.000, Y  +660.593, Z    +0.000, E1   -32.163, E3 +147971.875}
SPL {X  -160.000, Y  +665.836, Z    +0.000, E1   -32.154, E3 +147989.592}
SPL {X  -160.000, Y  +670.613, Z    +0.000, E1   -32.138, E3 +148005.802}
SPL {X  -159.954, Y  +675.336, Z    +0.000, E1   -32.135, E3 +148021.810}
SPL {X  -159.758, Y  +680.302, Z    +0.000, E1   -32.108, E3 +148038.825}
SPL {X  -159.416, Y  +685.158, Z    +0.000, E1   -32.039, E3 +148055.636}
SPL {X  -158.953, Y  +689.772, Z    +0.000, E1   -31.965, E3 +148071.736}
SPL {X  -158.363, Y  +694.328, Z    +0.000, E1   -31.871, E3 +148087.748}
SPL {X  -157.606, Y  +699.074, Z    +0.000, E1   -31.756, E3 +148104.592}
SPL {X  -156.791, Y  +703.384, Z    +0.000, E1   -31.607, E3 +148120.042}
SPL {X  -155.792, Y  +707.952, Z    +0.000, E1   -31.465, E3 +148136.488}
SPL {X  -155.149, Y  +710.598, Z    +0.000, E1   -26.183, E3 +148191.948}
ENDSPLINE

SPLINE
SPL {X  -158.679, Y  +692.020, Z    +0.000, E1   -14.212, E3 +148225.624}
SPL {X  -159.747, Y  +680.500, Z    +0.000, E1    -7.378, E3 +148234.002}
SPL {X  -160.000, Y  +671.618, Z    +0.000, E1    -1.592, E3 +148237.616}
SPL {X  -160.000, Y  +666.041, Z    +0.000, E1    +2.615, E3 +148239.583}
SPL {X  -160.000, Y  +661.396, Z    +0.000, E1    +6.484, E3 +148241.256}
SPL {X  -160.000, Y  +653.532, Z    +0.000, E1   +13.136, E3 +148245.376}
SPL {X  -160.000, Y  +631.927, Z    +0.000, E1   +26.832, E3 +148268.143}
SPL {X  -160.000, Y  +610.736, Z    +0.000, E1   +32.114, E3 +148310.812}
SPL {X  -160.000, Y  +605.907, Z    +0.000, E1   +32.114, E3 +148327.161}
SPL {X  -160.000, Y  +601.221, Z    +0.000, E1   +32.108, E3 +148343.028}
SPL {X  -160.000, Y  +596.433, Z    +0.000, E1   +32.120, E3 +148359.210}
SPL {X  -160.000, Y  +592.025, Z    +0.000, E1   +32.104, E3 +148374.135}
SPL {X  -160.000, Y  +587.734, Z    +0.000, E1   +32.110, E3 +148388.655}
SPL {X  -160.000, Y  +583.150, Z    +0.000, E1   +32.111, E3 +148404.182}
SPL {X  -160.000, Y  +579.063, Z    +0.000, E1   +32.085, E3 +148418.084}
SPL {X  -160.000, Y  +574.897, Z    +0.000, E1   +32.110, E3 +148432.135}
SPL {X  -160.000, Y  +570.471, Z    +0.000, E1   +32.093, E3 +148447.150}
SPL {X  -160.000, Y  +566.667, Z    +0.000, E1   +32.086, E3 +148460.064}
SPL {X  -160.000, Y  +562.434, Z    +0.000, E1   +32.097, E3 +148474.374}
SPL {X  -160.000, Y  +557.710, Z    +0.000, E1   +32.104, E3 +148490.357}
SPL {X  -160.000, Y  +553.479, Z    +0.000, E1   +32.081, E3 +148504.726}
SPL {X  -160.000, Y  +547.489, Z    +0.000, E1   +32.181, E3 +148524.845}
SPL {X  -160.000, Y  +541.554, Z    +0.000, E1   +32.092, E3 +148545.082}
SPL {X  -160.000, Y  +537.332, Z    +0.000, E1   +32.092, E3 +148559.379}
SPL {X  -160.000, Y  +533.113, Z    +0.000, E1   +32.090, E3 +148573.676}
SPL {X  -160.000, Y  +528.875, Z    +0.000, E1   +32.090, E3 +148588.019}
SPL {X  -160.000, Y  +524.453, Z    +0.000, E1   +32.104, E3 +148602.943}
SPL {X  -160.000, Y  +520.037, Z    +0.000, E1   +32.096, E3 +148617.885}
SPL {X  -160.000, Y  +514.030, Z    +0.000, E1   +32.182, E3 +148638.081}
SPL {X  -160.000, Y  +508.131, Z    +0.000, E1   +32.099, E3 +148658.186}
SPL {X  -160.000, Y  +504.077, Z    +0.000, E1   +32.094, E3 +148671.909}
SPL {X  -160.000, Y  +494.657, Z    +0.000, E1   +34.509, E3 +148686.772}
SPL {X  -160.000, Y  +491.565, Z    +0.000, E1   +33.823, E3 +148700.679}
SPL {X  -160.000, Y  +489.317, Z    +0.000, E1   +32.894, E3 +148714.024}
SPL {X  -160.000, Y  +486.958, Z    +0.000, E1   +31.703, E3 +148729.795}
SPL {X  -160.000, Y  +484.144, Z    +0.000, E1   +30.999, E3 +148744.218}
SPL {X  -160.000, Y  +479.156, Z    +0.000, E1   +31.035, E3 +148761.784}
SPL {X  -160.000, Y  +474.045, Z    +0.000, E1   +31.015, E3 +148779.876}
SPL {X  -160.000, Y  +468.999, Z    +0.000, E1   +31.021, E3 +148797.701}
SPL {X  -160.000, Y  +464.107, Z    +0.000, E1   +31.012, E3 +148815.001}
SPL {X  -160.000, Y  +459.262, Z    +0.000, E1   +31.016, E3 +148832.108}
SPL {X  -160.000, Y  +454.119, Z    +0.000, E1   +31.026, E3 +148850.257}
SPL {X  -160.000, Y  +448.874, Z    +0.000, E1   +31.019, E3 +148868.813}
SPL {X  -160.000, Y  +443.892, Z    +0.000, E1   +31.019, E3 +148886.401}
SPL {X  -160.000, Y  +438.782, Z    +0.000, E1   +31.022, E3 +148904.476}
SPL {X  -160.000, Y  +433.722, Z    +0.000, E1   +31.007, E3 +148922.420}
SPL {X  -160.000, Y  +428.980, Z    +0.000, E1   +31.004, E3 +148939.177}
SPL {X  -160.000, Y  +424.339, Z    +0.000, E1   +31.006, E3 +148955.551}
SPL {X  -160.000, Y  +419.231, Z    +0.000, E1   +31.030, E3 +148973.545}
SPL {X  -160.000, Y  +414.179, Z    +0.000, E1   +31.008, E3 +148991.442}
SPL {X  -160.000, Y  +409.416, Z    +0.000, E1   +31.023, E3 +149008.225}
SPL {X  -160.000, Y  +403.994, Z    +0.000, E1   +31.033, E3 +149027.381}
SPL {X  -160.000, Y  +399.052, Z    +0.000, E1   +31.010, E3 +149044.849}
SPL {X  -160.000, Y  +394.012, Z    +0.000, E1   +31.036, E3 +149062.637}
SPL {X  -159.999, Y  +388.376, Z    +0.000, E1   +31.028, E3 +149082.567}
SPL {X  -159.897, Y  +383.070, Z    +0.000, E1   +31.010, E3 +149101.405}
SPL {X  -159.656, Y  +378.313, Z    +0.000, E1   +30.961, E3 +149118.497}
SPL {X  -159.237, Y  +373.190, Z    +0.000, E1   +30.917, E3 +149136.998}
SPL {X  -158.628, Y  +367.891, Z    +0.000, E1   +30.812, E3 +149156.383}
SPL {X  -157.915, Y  +363.053, Z    +0.000, E1   +30.689, E3 +149174.250}
SPL {X  -157.216, Y  +359.084, Z    +0.000, E1   +30.550, E3 +149189.053}
SPL {X  -156.248, Y  +354.355, Z    +0.000, E1   +30.460, E3 +149206.665}
SPL {X  -155.629, Y  +351.657, Z    +0.000, E1   +25.972, E3 +149253.094}
ENDSPLINE

SPLINE
SPL {X  -156.240, Y  +354.319, Z    +0.000, E1   +23.538, E3 +149265.701}
SPL {X  -159.137, Y  +372.201, Z    +0.000, E1   +12.017, E3 +149295.538}
SPL {X  -159.858, Y  +382.069, Z    +0.000, E1    +5.945, E3 +149302.056}
SPL {X  -160.000, Y  +389.339, Z    +0.000, E1    +1.101, E3 +149305.218}
SPL {X  -160.000, Y  +395.749, Z    +0.000, E1    -3.722, E3 +149307.824}
SPL {X  -160.000, Y  +403.128, Z    +0.000, E1    -9.899, E3 +149311.128}
SPL {X  -160.000, Y  +411.609, Z    +0.000, E1   -16.851, E3 +149316.449}
SPL {X  -160.000, Y  +429.715, Z    +0.000, E1   -27.376, E3 +149335.812}
SPL {X  -160.000, Y  +449.791, Z    +0.000, E1   -32.145, E3 +149377.049}
SPL {X  -160.000, Y  +454.903, Z    +0.000, E1   -32.134, E3 +149394.354}
SPL {X  -160.000, Y  +460.041, Z    +0.000, E1   -32.144, E3 +149411.707}
SPL {X  -160.000, Y  +465.466, Z    +0.000, E1   -32.152, E3 +149430.025}
SPL {X  -160.000, Y  +471.112, Z    +0.000, E1   -32.154, E3 +149449.113}
SPL {X  -160.000, Y  +476.735, Z    +0.000, E1   -32.156, E3 +149468.104}
SPL {X  -160.000, Y  +482.675, Z    +0.000, E1   -32.169, E3 +149488.153}
SPL {X  -160.000, Y  +488.008, Z    +0.000, E1   -32.144, E3 +149506.199}
SPL {X  -160.000, Y  +493.245, Z    +0.000, E1   -32.159, E3 +149523.908}
SPL {X  -160.000, Y  +498.210, Z    +0.000, E1   -32.128, E3 +149540.742}
SPL {X  -160.000, Y  +503.407, Z    +0.000, E1   -32.165, E3 +149558.246}
SPL {X  -160.000, Y  +509.142, Z    +0.000, E1   -32.157, E3 +149577.641}
SPL {X  -160.000, Y  +514.696, Z    +0.000, E1   -32.156, E3 +149596.422}
SPL {X  -160.000, Y  +520.339, Z    +0.000, E1   -32.159, E3 +149615.494}
SPL {X  -160.000, Y  +525.825, Z    +0.000, E1   -32.148, E3 +149634.058}
SPL {X  -160.000, Y  +530.379, Z    +0.000, E1   -32.130, E3 +149649.486}
SPL {X  -160.000, Y  +535.020, Z    +0.000, E1   -32.146, E3 +149665.132}
SPL {X  -160.000, Y  +540.303, Z    +0.000, E1   -32.158, E3 +149682.957}
SPL {X  -160.000, Y  +545.740, Z    +0.000, E1   -32.155, E3 +149701.350}
SPL {X  -160.000, Y  +550.807, Z    +0.000, E1   -32.147, E3 +149718.473}
SPL {X  -160.000, Y  +555.841, Z    +0.000, E1   -32.148, E3 +149735.512}
SPL {X  -160.000, Y  +561.018, Z    +0.000, E1   -32.143, E3 +149753.041}
SPL {X  -160.000, Y  +566.466, Z    +0.000, E1   -32.153, E3 +149771.459}
SPL {X  -160.000, Y  +571.733, Z    +0.000, E1   -32.135, E3 +149789.296}
SPL {X  -160.000, Y  +576.943, Z    +0.000, E1   -32.148, E3 +149806.892}
SPL {X  -160.000, Y  +582.183, Z    +0.000, E1   -32.140, E3 +149824.617}
SPL {X  -160.000, Y  +587.036, Z    +0.000, E1   -32.141, E3 +149840.988}
SPL {X  -160.000, Y  +591.785, Z    +0.000, E1   -32.144, E3 +149857.012}
SPL {X  -160.000, Y  +596.962, Z    +0.000, E1   -32.161, E3 +149874.498}
SPL {X  -160.000, Y  +601.800, Z    +0.000, E1   -32.134, E3 +149890.895}
SPL {X  -160.000, Y  +606.611, Z    +0.000, E1   -32.156, E3 +149907.110}
SPL {X  -160.000, Y  +611.219, Z    +0.000, E1   -32.131, E3 +149922.723}
SPL {X  -160.000, Y  +616.331, Z    +0.000, E1   -32.174, E3 +149939.921}
SPL {X  -160.000, Y  +621.751, Z    +0.000, E1   -32.150, E3 +149958.263}
SPL {X  -160.000, Y  +626.312, Z    +0.000, E1   -32.145, E3 +149973.669}
SPL {X  -160.000, Y  +630.971, Z    +0.000, E1   -32.155, E3 +149989.397}
SPL {X  -160.000, Y  +635.550, Z    +0.000, E1   -32.137, E3 +150004.923}
SPL {X  -160.000, Y  +640.419, Z    +0.000, E1   -32.158, E3 +150021.361}
SPL {X  -160.000, Y  +645.749, Z    +0.000, E1   -32.151, E3 +150039.387}
SPL {X  -160.000, Y  +650.662, Z    +0.000, E1   -32.150, E3 +150055.958}
SPL {X  -160.000, Y  +655.372, Z    +0.000, E1   -32.145, E3 +150071.905}
SPL {X  -160.000, Y  +660.593, Z    +0.000, E1   -32.163, E3 +150089.522}
SPL {X  -160.000, Y  +665.836, Z    +0.000, E1   -32.154, E3 +150107.239}
SPL {X  -160.000, Y  +670.613, Z    +0.000, E1   -32.138, E3 +150123.449}
SPL {X  -159.954, Y  +675.336, Z    +0.000, E1   -32.135, E3 +150139.458}
SPL {X  -159.758, Y  +680.302, Z    +0.000, E1   -32.108, E3 +150156.472}
SPL {X  -159.416, Y  +685.158, Z    +0.000, E1   -32.039, E3 +150173.284}
SPL {X  -158.953, Y  +689.772, Z    +0.000, E1   -31.965, E3 +150189.383}
SPL {X  -158.363, Y  +694.328, Z    +0.000, E1   -31.871, E3 +150205.396}
SPL {X  -157.606, Y  +699.074, Z    +0.000, E1   -31.756, E3 +150222.239}
SPL {X  -156.791, Y  +703.384, Z    +0.000, E1   -31.607, E3 +150237.689}
SPL {X  -155.792, Y  +707.952, Z    +0.000, E1   -31.465, E3 +150254.135}
SPL {X  -155.149, Y  +710.598, Z    +0.000, E1   -26.183, E3 +150309.595}
ENDSPLINE

SPLINE
SPL {X  -158.679, Y  +692.020, Z    +0.000, E1   -14.212, E3 +150343.272}
SPL {X  -159.747, Y  +680.500, Z    +0.000, E1    -7.378, E3 +150351.649}
SPL {X  -160.000, Y  +671.618, Z    +0.000, E1    -1.592, E3 +150355.264}
SPL {X  -160.000, Y  +666.041, Z    +0.000, E1    +2.615, E3 +150357.230}
SPL {X  -160.000, Y  +661.396, Z    +0.000, E1    +6.484, E3 +150358.903}
SPL {X  -160.000, Y  +653.532, Z    +0.000, E1   +13.136, E3 +150363.023}
SPL {X  -160.000, Y  +631.927, Z    +0.000, E1   +26.832, E3 +150385.790}
SPL {X  -160.000, Y  +610.736, Z    +0.000, E1   +32.114, E3 +150428.459}
SPL {X  -160.000, Y  +605.907, Z    +0.000, E1   +32.114, E3 +150444.808}
SPL {X  -160.000, Y  +601.221, Z    +0.000, E1   +32.108, E3 +150460.675}
SPL {X  -160.000, Y  +596.433, Z    +0.000, E1   +32.120, E3 +150476.857}
SPL {X  -160.000, Y  +592.025, Z    +0.000, E1   +32.104, E3 +150491.782}
SPL {X  -160.000, Y  +587.734, Z    +0.000, E1   +32.110, E3 +150506.302}
SPL {X  -160.000, Y  +583.150, Z    +0.000, E1   +32.111, E3 +150521.830}
SPL {X  -160.000, Y  +579.063, Z    +0.000, E1   +32.085, E3 +150535.731}
SPL {X  -160.000, Y  +574.897, Z    +0.000, E1   +32.110, E3 +150549.783}
SPL {X  -160.000, Y  +570.471, Z    +0.000, E1   +32.093, E3 +150564.797}
SPL {X  -160.000, Y  +566.667, Z    +0.000, E1   +32.086, E3 +150577.711}
SPL {X  -160.000, Y  +562.434, Z    +0.000, E1   +32.097, E3 +150592.021}
SPL {X  -160.000, Y  +557.710, Z    +0.000, E1   +32.104, E3 +150608.004}
SPL {X  -160.000, Y  +553.479, Z    +0.000, E1   +32.081, E3 +150622.374}
SPL {X  -160.000, Y  +547.489, Z    +0.000, E1   +32.181, E3 +150642.492}
SPL {X  -160.000, Y  +541.554, Z    +0.000, E1   +32.092, E3 +150662.729}
SPL {X  -160.000, Y  +537.332, Z    +0.000, E1   +32.092, E3 +150677.026}
SPL {X  -160.000, Y  +533.113, Z    +0.000, E1   +32.090, E3 +150691.323}
SPL {X  -160.000, Y  +528.875, Z    +0.000, E1   +32.090, E3 +150705.666}
SPL {X  -160.000, Y  +524.453, Z    +0.000, E1   +32.104, E3 +150720.590}
SPL {X  -160.000, Y  +520.037, Z    +0.000, E1   +32.096, E3 +150735.532}
SPL {X  -160.000, Y  +514.030, Z    +0.000, E1   +32.182, E3 +150755.728}
SPL {X  -160.000, Y  +508.131, Z    +0.000, E1   +32.099, E3 +150775.833}
SPL {X  -160.000, Y  +504.077, Z    +0.000, E1   +32.094, E3 +150789.556}
SPL {X  -160.000, Y  +494.657, Z    +0.000, E1   +34.509, E3 +150804.419}
SPL {X  -160.000, Y  +491.565, Z    +0.000, E1   +33.823, E3 +150818.326}
SPL {X  -160.000, Y  +489.317, Z    +0.000, E1   +32.894, E3 +150831.671}
SPL {X  -160.000, Y  +486.958, Z    +0.000, E1   +31.703, E3 +150847.443}
SPL {X  -160.000, Y  +484.144, Z    +0.000, E1   +30.999, E3 +150861.865}
SPL {X  -160.000, Y  +479.156, Z    +0.000, E1   +31.035, E3 +150879.431}
SPL {X  -160.000, Y  +474.045, Z    +0.000, E1   +31.015, E3 +150897.523}
SPL {X  -160.000, Y  +468.999, Z    +0.000, E1   +31.021, E3 +150915.348}
SPL {X  -160.000, Y  +464.107, Z    +0.000, E1   +31.012, E3 +150932.648}
SPL {X  -160.000, Y  +459.262, Z    +0.000, E1   +31.016, E3 +150949.755}
SPL {X  -160.000, Y  +454.119, Z    +0.000, E1   +31.026, E3 +150967.905}
SPL {X  -160.000, Y  +448.874, Z    +0.000, E1   +31.019, E3 +150986.461}
SPL {X  -160.000, Y  +443.892, Z    +0.000, E1   +31.019, E3 +151004.049}
SPL {X  -160.000, Y  +438.782, Z    +0.000, E1   +31.022, E3 +151022.123}
SPL {X  -160.000, Y  +433.722, Z    +0.000, E1   +31.007, E3 +151040.067}
SPL {X  -160.000, Y  +428.980, Z    +0.000, E1   +31.004, E3 +151056.824}
SPL {X  -160.000, Y  +424.339, Z    +0.000, E1   +31.006, E3 +151073.198}
SPL {X  -160.000, Y  +419.231, Z    +0.000, E1   +31.030, E3 +151091.192}
SPL {X  -160.000, Y  +414.179, Z    +0.000, E1   +31.008, E3 +151109.089}
SPL {X  -160.000, Y  +409.416, Z    +0.000, E1   +31.023, E3 +151125.872}
SPL {X  -160.000, Y  +403.994, Z    +0.000, E1   +31.033, E3 +151145.028}
SPL {X  -160.000, Y  +399.052, Z    +0.000, E1   +31.010, E3 +151162.496}
SPL {X  -160.000, Y  +394.012, Z    +0.000, E1   +31.036, E3 +151180.285}
SPL {X  -159.999, Y  +388.376, Z    +0.000, E1   +31.028, E3 +151200.214}
SPL {X  -159.897, Y  +383.070, Z    +0.000, E1   +31.010, E3 +151219.053}
SPL {X  -159.656, Y  +378.313, Z    +0.000, E1   +30.961, E3 +151236.145}
SPL {X  -159.237, Y  +373.190, Z    +0.000, E1   +30.917, E3 +151254.645}
SPL {X  -158.628, Y  +367.891, Z    +0.000, E1   +30.812, E3 +151274.031}
SPL {X  -157.915, Y  +363.053, Z    +0.000, E1   +30.689, E3 +151291.898}
SPL {X  -157.216, Y  +359.084, Z    +0.000, E1   +30.550, E3 +151306.700}
SPL {X  -156.248, Y  +354.355, Z    +0.000, E1   +30.460, E3 +151324.312}
SPL {X  -155.629, Y  +351.657, Z    +0.000, E1   +25.972, E3 +151370.741}
ENDSPLINE

SPLINE
SPL {X  -156.240, Y  +354.319, Z    +0.000, E1   +23.538, E3 +151383.349}
SPL {X  -159.137, Y  +372.201, Z    +0.000, E1   +12.017, E3 +151413.186}
SPL {X  -159.858, Y  +382.069, Z    +0.000, E1    +5.945, E3 +151419.703}
SPL {X  -160.000, Y  +389.339, Z    +0.000, E1    +1.101, E3 +151422.866}
SPL {X  -160.000, Y  +395.749, Z    +0.000, E1    -3.722, E3 +151425.471}
SPL {X  -160.000, Y  +403.128, Z    +0.000, E1    -9.899, E3 +151428.775}
SPL {X  -160.000, Y  +411.609, Z    +0.000, E1   -16.851, E3 +151434.096}
SPL {X  -160.000, Y  +429.715, Z    +0.000, E1   -27.376, E3 +151453.460}
SPL {X  -160.000, Y  +449.791, Z    +0.000, E1   -32.145, E3 +151494.697}
SPL {X  -160.000, Y  +454.903, Z    +0.000, E1   -32.134, E3 +151512.001}
SPL {X  -160.000, Y  +460.041, Z    +0.000, E1   -32.144, E3 +151529.354}
SPL {X  -160.000, Y  +465.466, Z    +0.000, E1   -32.152, E3 +151547.672}
SPL {X  -160.000, Y  +471.112, Z    +0.000, E1   -32.154, E3 +151566.760}
SPL {X  -160.000, Y  +476.735, Z    +0.000, E1   -32.156, E3 +151585.751}
SPL {X  -160.000, Y  +482.675, Z    +0.000, E1   -32.169, E3 +151605.800}
SPL {X  -160.000, Y  +488.008, Z    +0.000, E1   -32.144, E3 +151623.846}
SPL {X  -160.000, Y  +493.245, Z    +0.000, E1   -32.159, E3 +151641.555}
SPL {X  -160.000, Y  +498.210, Z    +0.000, E1   -32.128, E3 +151658.389}
SPL {X  -160.000, Y  +503.407, Z    +0.000, E1   -32.165, E3 +151675.893}
SPL {X  -160.000, Y  +509.142, Z    +0.000, E1   -32.157, E3 +151695.289}
SPL {X  -160.000, Y  +514.696, Z    +0.000, E1   -32.156, E3 +151714.069}
SPL {X  -160.000, Y  +520.339, Z    +0.000, E1   -32.159, E3 +151733.141}
SPL {X  -160.000, Y  +525.825, Z    +0.000, E1   -32.148, E3 +151751.705}
SPL {X  -160.000, Y  +530.379, Z    +0.000, E1   -32.130, E3 +151767.133}
SPL {X  -160.000, Y  +535.020, Z    +0.000, E1   -32.146, E3 +151782.779}
SPL {X  -160.000, Y  +540.303, Z    +0.000, E1   -32.158, E3 +151800.604}
SPL {X  -160.000, Y  +545.740, Z    +0.000, E1   -32.155, E3 +151818.997}
SPL {X  -160.000, Y  +550.807, Z    +0.000, E1   -32.147, E3 +151836.120}
SPL {X  -160.000, Y  +555.841, Z    +0.000, E1   -32.148, E3 +151853.159}
SPL {X  -160.000, Y  +561.018, Z    +0.000, E1   -32.143, E3 +151870.688}
SPL {X  -160.000, Y  +566.466, Z    +0.000, E1   -32.153, E3 +151889.106}
SPL {X  -160.000, Y  +571.733, Z    +0.000, E1   -32.135, E3 +151906.943}
SPL {X  -160.000, Y  +576.943, Z    +0.000, E1   -32.148, E3 +151924.540}
SPL {X  -160.000, Y  +582.183, Z    +0.000, E1   -32.140, E3 +151942.264}
SPL {X  -160.000, Y  +587.036, Z    +0.000, E1   -32.141, E3 +151958.635}
SPL {X  -160.000, Y  +591.785, Z    +0.000, E1   -32.144, E3 +151974.659}
SPL {X  -160.000, Y  +596.962, Z    +0.000, E1   -32.161, E3 +151992.145}
SPL {X  -160.000, Y  +601.800, Z    +0.000, E1   -32.134, E3 +152008.543}
SPL {X  -160.000, Y  +606.611, Z    +0.000, E1   -32.156, E3 +152024.757}
SPL {X  -160.000, Y  +611.219, Z    +0.000, E1   -32.131, E3 +152040.370}
SPL {X  -160.000, Y  +616.331, Z    +0.000, E1   -32.174, E3 +152057.568}
SPL {X  -160.000, Y  +621.751, Z    +0.000, E1   -32.150, E3 +152075.911}
SPL {X  -160.000, Y  +626.312, Z    +0.000, E1   -32.145, E3 +152091.317}
SPL {X  -160.000, Y  +630.971, Z    +0.000, E1   -32.155, E3 +152107.045}
SPL {X  -160.000, Y  +635.550, Z    +0.000, E1   -32.137, E3 +152122.571}
SPL {X  -160.000, Y  +640.419, Z    +0.000, E1   -32.158, E3 +152139.009}
SPL {X  -160.000, Y  +645.749, Z    +0.000, E1   -32.151, E3 +152157.034}
SPL {X  -160.000, Y  +650.662, Z    +0.000, E1   -32.150, E3 +152173.605}
SPL {X  -160.000, Y  +655.372, Z    +0.000, E1   -32.145, E3 +152189.552}
SPL {X  -160.000, Y  +660.593, Z    +0.000, E1   -32.163, E3 +152207.170}
SPL {X  -160.000, Y  +665.836, Z    +0.000, E1   -32.154, E3 +152224.886}
SPL {X  -160.000, Y  +670.613, Z    +0.000, E1   -32.138, E3 +152241.097}
SPL {X  -159.954, Y  +675.336, Z    +0.000, E1   -32.135, E3 +152257.105}
SPL {X  -159.758, Y  +680.302, Z    +0.000, E1   -32.108, E3 +152274.120}
SPL {X  -159.416, Y  +685.158, Z    +0.000, E1   -32.039, E3 +152290.931}
SPL {X  -158.953, Y  +689.772, Z    +0.000, E1   -31.965, E3 +152307.030}
SPL {X  -158.363, Y  +694.328, Z    +0.000, E1   -31.871, E3 +152323.043}
SPL {X  -157.606, Y  +699.074, Z    +0.000, E1   -31.756, E3 +152339.886}
SPL {X  -156.791, Y  +703.384, Z    +0.000, E1   -31.607, E3 +152355.336}
SPL {X  -155.792, Y  +707.952, Z    +0.000, E1   -31.465, E3 +152371.783}
SPL {X  -155.149, Y  +710.598, Z    +0.000, E1   -26.183, E3 +152427.243}
ENDSPLINE

SPLINE
SPL {X  -158.679, Y  +692.020, Z    +0.000, E1   -14.212, E3 +152460.919}
SPL {X  -159.747, Y  +680.500, Z    +0.000, E1    -7.378, E3 +152469.297}
SPL {X  -160.000, Y  +671.618, Z    +0.000, E1    -1.592, E3 +152472.911}
SPL {X  -160.000, Y  +666.041, Z    +0.000, E1    +2.615, E3 +152474.878}
SPL {X  -160.000, Y  +661.396, Z    +0.000, E1    +6.484, E3 +152476.550}
SPL {X  -160.000, Y  +653.532, Z    +0.000, E1   +13.136, E3 +152480.671}
SPL {X  -160.000, Y  +631.927, Z    +0.000, E1   +26.832, E3 +152503.437}
SPL {X  -160.000, Y  +610.736, Z    +0.000, E1   +32.114, E3 +152546.107}
SPL {X  -160.000, Y  +605.907, Z    +0.000, E1   +32.114, E3 +152562.455}
SPL {X  -160.000, Y  +601.221, Z    +0.000, E1   +32.108, E3 +152578.323}
SPL {X  -160.000, Y  +596.433, Z    +0.000, E1   +32.120, E3 +152594.505}
SPL {X  -160.000, Y  +592.025, Z    +0.000, E1   +32.104, E3 +152609.429}
SPL {X  -160.000, Y  +587.734, Z    +0.000, E1   +32.110, E3 +152623.950}
SPL {X  -160.000, Y  +583.150, Z    +0.000, E1   +32.111, E3 +152639.477}
SPL {X  -160.000, Y  +579.063, Z    +0.000, E1   +32.085, E3 +152653.378}
SPL {X  -160.000, Y  +574.897, Z    +0.000, E1   +32.110, E3 +152667.430}
SPL {X  -160.000, Y  +570.471, Z    +0.000, E1   +32.093, E3 +152682.444}
SPL {X  -160.000, Y  +566.667, Z    +0.000, E1   +32.086, E3 +152695.359}
SPL {X  -160.000, Y  +562.434, Z    +0.000, E1   +32.097, E3 +152709.668}
SPL {X  -160.000, Y  +557.710, Z    +0.000, E1   +32.104, E3 +152725.652}
SPL {X  -160.000, Y  +553.479, Z    +0.000, E1   +32.081, E3 +152740.021}
SPL {X  -160.000, Y  +547.489, Z    +0.000, E1   +32.181, E3 +152760.139}
SPL {X  -160.000, Y  +541.554, Z    +0.000, E1   +32.092, E3 +152780.376}
SPL {X  -160.000, Y  +537.332, Z    +0.000, E1   +32.092, E3 +152794.674}
SPL {X  -160.000, Y  +533.113, Z    +0.000, E1   +32.090, E3 +152808.970}
SPL {X  -160.000, Y  +528.875, Z    +0.000, E1   +32.090, E3 +152823.314}
SPL {X  -160.000, Y  +524.453, Z    +0.000, E1   +32.104, E3 +152838.238}
SPL {X  -160.000, Y  +520.037, Z    +0.000, E1   +32.096, E3 +152853.180}
SPL {X  -160.000, Y  +514.030, Z    +0.000, E1   +32.182, E3 +152873.376}
SPL {X  -160.000, Y  +508.131, Z    +0.000, E1   +32.099, E3 +152893.480}
SPL {X  -160.000, Y  +504.077, Z    +0.000, E1   +32.094, E3 +152907.203}
SPL {X  -160.000, Y  +494.657, Z    +0.000, E1   +34.509, E3 +152922.066}
SPL {X  -160.000, Y  +491.565, Z    +0.000, E1   +33.823, E3 +152935.973}
SPL {X  -160.000, Y  +489.317, Z    +0.000, E1   +32.894, E3 +152949.318}
SPL {X  -160.000, Y  +486.958, Z    +0.000, E1   +31.703, E3 +152965.090}
SPL {X  -160.000, Y  +484.144, Z    +0.000, E1   +30.999, E3 +152979.513}
SPL {X  -160.000, Y  +479.156, Z    +0.000, E1   +31.035, E3 +152997.079}
SPL {X  -160.000, Y  +474.045, Z    +0.000, E1   +31.015, E3 +153015.170}
SPL {X  -160.000, Y  +468.999, Z    +0.000, E1   +31.021, E3 +153032.996}
SPL {X  -160.000, Y  +464.107, Z    +0.000, E1   +31.012, E3 +153050.296}
SPL {X  -160.000, Y  +459.262, Z    +0.000, E1   +31.016, E3 +153067.403}
SPL {X  -160.000, Y  +454.119, Z    +0.000, E1   +31.026, E3 +153085.552}
SPL {X  -160.000, Y  +448.874, Z    +0.000, E1   +31.019, E3 +153104.108}
SPL {X  -160.000, Y  +443.892, Z    +0.000, E1   +31.019, E3 +153121.696}
SPL {X  -160.000, Y  +438.782, Z    +0.000, E1   +31.022, E3 +153139.770}
SPL {X  -160.000, Y  +433.722, Z    +0.000, E1   +31.007, E3 +153157.714}
SPL {X  -160.000, Y  +428.980, Z    +0.000, E1   +31.004, E3 +153174.471}
SPL {X  -160.000, Y  +424.339, Z    +0.000, E1   +31.006, E3 +153190.846}
SPL {X  -160.000, Y  +419.231, Z    +0.000, E1   +31.030, E3 +153208.839}
SPL {X  -160.000, Y  +414.179, Z    +0.000, E1   +31.008, E3 +153226.736}
SPL {X  -160.000, Y  +409.416, Z    +0.000, E1   +31.023, E3 +153243.520}
SPL {X  -160.000, Y  +403.994, Z    +0.000, E1   +31.033, E3 +153262.675}
SPL {X  -160.000, Y  +399.052, Z    +0.000, E1   +31.010, E3 +153280.143}
SPL {X  -160.000, Y  +394.012, Z    +0.000, E1   +31.036, E3 +153297.932}
SPL {X  -159.999, Y  +388.376, Z    +0.000, E1   +31.028, E3 +153317.862}
SPL {X  -159.897, Y  +383.070, Z    +0.000, E1   +31.010, E3 +153336.700}
SPL {X  -159.656, Y  +378.313, Z    +0.000, E1   +30.961, E3 +153353.792}
SPL {X  -159.237, Y  +373.190, Z    +0.000, E1   +30.917, E3 +153372.292}
SPL {X  -158.628, Y  +367.891, Z    +0.000, E1   +30.812, E3 +153391.678}
SPL {X  -157.915, Y  +363.053, Z    +0.000, E1   +30.689, E3 +153409.545}
SPL {X  -157.216, Y  +359.084, Z    +0.000, E1   +30.550, E3 +153424.347}
SPL {X  -156.248, Y  +354.355, Z    +0.000, E1   +30.460, E3 +153441.960}
SPL {X  -155.629, Y  +351.657, Z    +0.000, E1   +25.972, E3 +153488.388}
ENDSPLINE

SPLINE
SPL {X  -156.240, Y  +354.319, Z    +0.000, E1   +23.538, E3 +153500.996}
SPL {X  -159.137, Y  +372.201, Z    +0.000, E1   +12.017, E3 +153530.833}
SPL {X  -159.858, Y  +382.069, Z    +0.000, E1    +5.945, E3 +153537.351}
SPL {X  -160.000, Y  +389.339, Z    +0.000, E1    +1.101, E3 +153540.513}
SPL {X  -160.000, Y  +395.749, Z    +0.000, E1    -3.722, E3 +153543.118}
SPL {X  -160.000, Y  +403.128, Z    +0.000, E1    -9.899, E3 +153546.422}
SPL {X  -160.000, Y  +411.609, Z    +0.000, E1   -16.851, E3 +153551.743}
SPL {X  -160.000, Y  +429.715, Z    +0.000, E1   -27.376, E3 +153571.107}
SPL {X  -160.000, Y  +449.791, Z    +0.000, E1   -32.145, E3 +153612.344}
SPL {X  -160.000, Y  +454.903, Z    +0.000, E1   -32.134, E3 +153629.648}
SPL {X  -160.000, Y  +460.041, Z    +0.000, E1   -32.144, E3 +153647.002}
SPL {X  -160.000, Y  +465.466, Z    +0.000, E1   -32.152, E3 +153665.319}
SPL {X  -160.000, Y  +471.112, Z    +0.000, E1   -32.154, E3 +153684.408}
SPL {X  -160.000, Y  +476.735, Z    +0.000, E1   -32.156, E3 +153703.399}
SPL {X  -160.000, Y  +482.675, Z    +0.000, E1   -32.169, E3 +153723.447}
SPL {X  -160.000, Y  +488.008, Z    +0.000, E1   -32.144, E3 +153741.494}
SPL {X  -160.000, Y  +493.245, Z    +0.000, E1   -32.159, E3 +153759.202}
SPL {X  -160.000, Y  +498.210, Z    +0.000, E1   -32.128, E3 +153776.037}
SPL {X  -160.000, Y  +503.407, Z    +0.000, E1   -32.165, E3 +153793.540}
SPL {X  -160.000, Y  +509.142, Z    +0.000, E1   -32.157, E3 +153812.936}
SPL {X  -160.000, Y  +514.696, Z    +0.000, E1   -32.156, E3 +153831.717}
SPL {X  -160.000, Y  +520.339, Z    +0.000, E1   -32.159, E3 +153850.789}
SPL {X  -160.000, Y  +525.825, Z    +0.000, E1   -32.148, E3 +153869.352}
SPL {X  -160.000, Y  +530.379, Z    +0.000, E1   -32.130, E3 +153884.780}
SPL {X  -160.000, Y  +535.020, Z    +0.000, E1   -32.146, E3 +153900.426}
SPL {X  -160.000, Y  +540.303, Z    +0.000, E1   -32.158, E3 +153918.252}
SPL {X  -160.000, Y  +545.740, Z    +0.000, E1   -32.155, E3 +153936.645}
SPL {X  -160.000, Y  +550.807, Z    +0.000, E1   -32.147, E3 +153953.767}
SPL {X  -160.000, Y  +555.841, Z    +0.000, E1   -32.148, E3 +153970.807}
SPL {X  -160.000, Y  +561.018, Z    +0.000, E1   -32.143, E3 +153988.335}
SPL {X  -160.000, Y  +566.466, Z    +0.000, E1   -32.153, E3 +154006.753}
SPL {X  -160.000, Y  +571.733, Z    +0.000, E1   -32.135, E3 +154024.590}
SPL {X  -160.000, Y  +576.943, Z    +0.000, E1   -32.148, E3 +154042.187}
SPL {X  -160.000, Y  +582.183, Z    +0.000, E1   -32.140, E3 +154059.912}
SPL {X  -160.000, Y  +587.036, Z    +0.000, E1   -32.141, E3 +154076.282}
SPL {X  -160.000, Y  +591.785, Z    +0.000, E1   -32.144, E3 +154092.306}
SPL {X  -160.000, Y  +596.962, Z    +0.000, E1   -32.161, E3 +154109.793}
SPL {X  -160.000, Y  +601.800, Z    +0.000, E1   -32.134, E3 +154126.190}
SPL {X  -160.000, Y  +606.611, Z    +0.000, E1   -32.156, E3 +154142.404}
SPL {X  -160.000, Y  +611.219, Z    +0.000, E1   -32.131, E3 +154158.018}
SPL {X  -160.000, Y  +616.331, Z    +0.000, E1   -32.174, E3 +154175.215}
SPL {X  -160.000, Y  +621.751, Z    +0.000, E1   -32.150, E3 +154193.558}
SPL {X  -160.000, Y  +626.312, Z    +0.000, E1   -32.145, E3 +154208.964}
SPL {X  -160.000, Y  +630.971, Z    +0.000, E1   -32.155, E3 +154224.692}
SPL {X  -160.000, Y  +635.550, Z    +0.000, E1   -32.137, E3 +154240.218}
SPL {X  -160.000, Y  +640.419, Z    +0.000, E1   -32.158, E3 +154256.656}
SPL {X  -160.000, Y  +645.749, Z    +0.000, E1   -32.151, E3 +154274.681}
SPL {X  -160.000, Y  +650.662, Z    +0.000, E1   -32.150, E3 +154291.253}
SPL {X  -160.000, Y  +655.372, Z    +0.000, E1   -32.145, E3 +154307.199}
SPL {X  -160.000, Y  +660.593, Z    +0.000, E1   -32.163, E3 +154324.817}
SPL {X  -160.000, Y  +665.836, Z    +0.000, E1   -32.154, E3 +154342.534}
SPL {X  -160.000, Y  +670.613, Z    +0.000, E1   -32.138, E3 +154358.744}
SPL {X  -159.954, Y  +675.336, Z    +0.000, E1   -32.135, E3 +154374.752}
SPL {X  -159.758, Y  +680.302, Z    +0.000, E1   -32.108, E3 +154391.767}
SPL {X  -159.416, Y  +685.158, Z    +0.000, E1   -32.039, E3 +154408.578}
SPL {X  -158.953, Y  +689.772, Z    +0.000, E1   -31.965, E3 +154424.678}
SPL {X  -158.363, Y  +694.328, Z    +0.000, E1   -31.871, E3 +154440.690}
SPL {X  -157.606, Y  +699.074, Z    +0.000, E1   -31.756, E3 +154457.533}
SPL {X  -156.791, Y  +703.384, Z    +0.000, E1   -31.607, E3 +154472.984}
SPL {X  -155.792, Y  +707.952, Z    +0.000, E1   -31.465, E3 +154489.430}
SPL {X  -155.149, Y  +710.598, Z    +0.000, E1   -26.183, E3 +154544.890}
ENDSPLINE

SPLINE
SPL {X  -158.679, Y  +692.020, Z    +0.000, E1   -14.212, E3 +154578.566}
SPL {X  -159.747, Y  +680.500, Z    +0.000, E1    -7.378, E3 +154586.944}
SPL {X  -160.000, Y  +671.618, Z    +0.000, E1    -1.592, E3 +154590.558}
SPL {X  -160.000, Y  +666.041, Z    +0.000, E1    +2.615, E3 +154592.525}
SPL {X  -160.000, Y  +661.396, Z    +0.000, E1    +6.484, E3 +154594.198}
SPL {X  -160.000, Y  +653.532, Z    +0.000, E1   +13.136, E3 +154598.318}
SPL {X  -160.000, Y  +631.927, Z    +0.000, E1   +26.832, E3 +154621.085}
SPL {X  -160.000, Y  +610.736, Z    +0.000, E1   +32.114, E3 +154663.754}
SPL {X  -160.000, Y  +605.907, Z    +0.000, E1   +32.114, E3 +154680.102}
SPL {X  -160.000, Y  +601.221, Z    +0.000, E1   +32.108, E3 +154695.970}
SPL {X  -160.000, Y  +596.433, Z    +0.000, E1   +32.120, E3 +154712.152}
SPL {X  -160.000, Y  +592.025, Z    +0.000, E1   +32.104, E3 +154727.077}
SPL {X  -160.000, Y  +587.734, Z    +0.000, E1   +32.110, E3 +154741.597}
SPL {X  -160.000, Y  +583.150, Z    +0.000, E1   +32.111, E3 +154757.124}
SPL {X  -160.000, Y  +579.063, Z    +0.000, E1   +32.085, E3 +154771.026}
SPL {X  -160.000, Y  +574.897, Z    +0.000, E1   +32.110, E3 +154785.077}
SPL {X  -160.000, Y  +570.471, Z    +0.000, E1   +32.093, E3 +154800.091}
SPL {X  -160.000, Y  +566.667, Z    +0.000, E1   +32.086, E3 +154813.006}
SPL {X  -160.000, Y  +562.434, Z    +0.000, E1   +32.097, E3 +154827.316}
SPL {X  -160.000, Y  +557.710, Z    +0.000, E1   +32.104, E3 +154843.299}
SPL {X  -160.000, Y  +553.479, Z    +0.000, E1   +32.081, E3 +154857.668}
SPL {X  -160.000, Y  +547.489, Z    +0.000, E1   +32.181, E3 +154877.787}
SPL {X  -160.000, Y  +541.554, Z    +0.000, E1   +32.092, E3 +154898.024}
SPL {X  -160.000, Y  +537.332, Z    +0.000, E1   +32.092, E3 +154912.321}
SPL {X  -160.000, Y  +533.113, Z    +0.000, E1   +32.090, E3 +154926.618}
SPL {X  -160.000, Y  +528.875, Z    +0.000, E1   +32.090, E3 +154940.961}
SPL {X  -160.000, Y  +524.453, Z    +0.000, E1   +32.104, E3 +154955.885}
SPL {X  -160.000, Y  +520.037, Z    +0.000, E1   +32.096, E3 +154970.827}
SPL {X  -160.000, Y  +514.030, Z    +0.000, E1   +32.182, E3 +154991.023}
SPL {X  -160.000, Y  +508.131, Z    +0.000, E1   +32.099, E3 +155011.128}
SPL {X  -160.000, Y  +504.077, Z    +0.000, E1   +32.094, E3 +155024.850}
SPL {X  -160.000, Y  +494.657, Z    +0.000, E1   +34.509, E3 +155039.713}
SPL {X  -160.000, Y  +491.565, Z    +0.000, E1   +33.823, E3 +155053.621}
SPL {X  -160.000, Y  +489.317, Z    +0.000, E1   +32.894, E3 +155066.966}
SPL {X  -160.000, Y  +486.958, Z    +0.000, E1   +31.703, E3 +155082.737}
SPL {X  -160.000, Y  +484.144, Z    +0.000, E1   +30.999, E3 +155097.160}
SPL {X  -160.000, Y  +479.156, Z    +0.000, E1   +31.035, E3 +155114.726}
SPL {X  -160.000, Y  +474.045, Z    +0.000, E1   +31.015, E3 +155132.818}
SPL {X  -160.000, Y  +468.999, Z    +0.000, E1   +31.021, E3 +155150.643}
SPL {X  -160.000, Y  +464.107, Z    +0.000, E1   +31.012, E3 +155167.943}
SPL {X  -160.000, Y  +459.262, Z    +0.000, E1   +31.016, E3 +155185.050}
SPL {X  -160.000, Y  +454.119, Z    +0.000, E1   +31.026, E3 +155203.199}
SPL {X  -160.000, Y  +448.874, Z    +0.000, E1   +31.019, E3 +155221.755}
SPL {X  -160.000, Y  +443.892, Z    +0.000, E1   +31.019, E3 +155239.343}
SPL {X  -160.000, Y  +438.782, Z    +0.000, E1   +31.022, E3 +155257.418}
SPL {X  -160.000, Y  +433.722, Z    +0.000, E1   +31.007, E3 +155275.362}
SPL {X  -160.000, Y  +428.980, Z    +0.000, E1   +31.004, E3 +155292.119}
SPL {X  -160.000, Y  +424.339, Z    +0.000, E1   +31.006, E3 +155308.493}
SPL {X  -160.000, Y  +419.231, Z    +0.000, E1   +31.030, E3 +155326.487}
SPL {X  -160.000, Y  +414.179, Z    +0.000, E1   +31.008, E3 +155344.384}
SPL {X  -160.000, Y  +409.416, Z    +0.000, E1   +31.023, E3 +155361.167}
SPL {X  -160.000, Y  +403.994, Z    +0.000, E1   +31.033, E3 +155380.323}
SPL {X  -160.000, Y  +399.052, Z    +0.000, E1   +31.010, E3 +155397.791}
SPL {X  -160.000, Y  +394.012, Z    +0.000, E1   +31.036, E3 +155415.579}
SPL {X  -159.999, Y  +388.376, Z    +0.000, E1   +31.028, E3 +155435.509}
SPL {X  -159.897, Y  +383.070, Z    +0.000, E1   +31.010, E3 +155454.347}
SPL {X  -159.656, Y  +378.313, Z    +0.000, E1   +30.961, E3 +155471.439}
SPL {X  -159.237, Y  +373.190, Z    +0.000, E1   +30.917, E3 +155489.939}
SPL {X  -158.628, Y  +367.891, Z    +0.000, E1   +30.812, E3 +155509.325}
SPL {X  -157.915, Y  +363.053, Z    +0.000, E1   +30.689, E3 +155527.192}
SPL {X  -157.216, Y  +359.084, Z    +0.000, E1   +30.550, E3 +155541.995}
SPL {X  -156.248, Y  +354.355, Z    +0.000, E1   +30.460, E3 +155559.607}
SPL {X  -155.629, Y  +351.657, Z    +0.000, E1   +25.972, E3 +155606.035}
ENDSPLINE

SPLINE
SPL {X  -156.240, Y  +354.319, Z    +0.000, E1   +23.538, E3 +155618.643}
SPL {X  -159.137, Y  +372.201, Z    +0.000, E1   +12.017, E3 +155648.480}
SPL {X  -159.858, Y  +382.069, Z    +0.000, E1    +5.945, E3 +155654.998}
SPL {X  -160.000, Y  +389.339, Z    +0.000, E1    +1.101, E3 +155658.160}
SPL {X  -160.000, Y  +395.749, Z    +0.000, E1    -3.722, E3 +155660.766}
SPL {X  -160.000, Y  +403.128, Z    +0.000, E1    -9.899, E3 +155664.070}
SPL {X  -160.000, Y  +411.609, Z    +0.000, E1   -16.851, E3 +155669.391}
SPL {X  -160.000, Y  +429.715, Z    +0.000, E1   -27.376, E3 +155688.754}
SPL {X  -160.000, Y  +449.791, Z    +0.000, E1   -32.145, E3 +155729.991}
SPL {X  -160.000, Y  +454.903, Z    +0.000, E1   -32.134, E3 +155747.295}
SPL {X  -160.000, Y  +460.041, Z    +0.000, E1   -32.144, E3 +155764.649}
SPL {X  -160.000, Y  +465.466, Z    +0.000, E1   -32.152, E3 +155782.967}
SPL {X  -160.000, Y  +471.112, Z    +0.000, E1   -32.154, E3 +155802.055}
SPL {X  -160.000, Y  +476.735, Z    +0.000, E1   -32.156, E3 +155821.046}
SPL {X  -160.000, Y  +482.675, Z    +0.000, E1   -32.169, E3 +155841.095}
SPL {X  -160.000, Y  +488.008, Z    +0.000, E1   -32.144, E3 +155859.141}
SPL {X  -160.000, Y  +493.245, Z    +0.000, E1   -32.159, E3 +155876.849}
SPL {X  -160.000, Y  +498.210, Z    +0.000, E1   -32.128, E3 +155893.684}
SPL {X  -160.000, Y  +503.407, Z    +0.000, E1   -32.165, E3 +155911.188}
SPL {X  -160.000, Y  +509.142, Z    +0.000, E1   -32.157, E3 +155930.583}
SPL {X  -160.000, Y  +514.696, Z    +0.000, E1   -32.156, E3 +155949.364}
SPL {X  -160.000, Y  +520.339, Z    +0.000, E1   -32.159, E3 +155968.436}
SPL {X  -160.000, Y  +525.825, Z    +0.000, E1   -32.148, E3 +155987.000}
SPL {X  -160.000, Y  +530.379, Z    +0.000, E1   -32.130, E3 +156002.428}
SPL {X  -160.000, Y  +535.020, Z    +0.000, E1   -32.146, E3 +156018.074}
SPL {X  -160.000, Y  +540.303, Z    +0.000, E1   -32.158, E3 +156035.899}
SPL {X  -160.000, Y  +545.740, Z    +0.000, E1   -32.155, E3 +156054.292}
SPL {X  -160.000, Y  +550.807, Z    +0.000, E1   -32.147, E3 +156071.414}
SPL {X  -160.000, Y  +555.841, Z    +0.000, E1   -32.148, E3 +156088.454}
SPL {X  -160.000, Y  +561.018, Z    +0.000, E1   -32.143, E3 +156105.983}
SPL {X  -160.000, Y  +566.466, Z    +0.000, E1   -32.153, E3 +156124.401}
SPL {X  -160.000, Y  +571.733, Z    +0.000, E1   -32.135, E3 +156142.237}
SPL {X  -160.000, Y  +576.943, Z    +0.000, E1   -32.148, E3 +156159.834}
SPL {X  -160.000, Y  +582.183, Z    +0.000, E1   -32.140, E3 +156177.559}
SPL {X  -160.000, Y  +587.036, Z    +0.000, E1   -32.141, E3 +156193.930}
SPL {X  -160.000, Y  +591.785, Z    +0.000, E1   -32.144, E3 +156209.953}
SPL {X  -160.000, Y  +596.962, Z    +0.000, E1   -32.161, E3 +156227.440}
SPL {X  -160.000, Y  +601.800, Z    +0.000, E1   -32.134, E3 +156243.837}
SPL {X  -160.000, Y  +606.611, Z    +0.000, E1   -32.156, E3 +156260.052}
SPL {X  -160.000, Y  +611.219, Z    +0.000, E1   -32.131, E3 +156275.665}
SPL {X  -160.000, Y  +616.331, Z    +0.000, E1   -32.174, E3 +156292.863}
SPL {X  -160.000, Y  +621.751, Z    +0.000, E1   -32.150, E3 +156311.205}
SPL {X  -160.000, Y  +626.312, Z    +0.000, E1   -32.145, E3 +156326.611}
SPL {X  -160.000, Y  +630.971, Z    +0.000, E1   -32.155, E3 +156342.339}
SPL {X  -160.000, Y  +635.550, Z    +0.000, E1   -32.137, E3 +156357.865}
SPL {X  -160.000, Y  +640.419, Z    +0.000, E1   -32.158, E3 +156374.303}
SPL {X  -160.000, Y  +645.749, Z    +0.000, E1   -32.151, E3 +156392.329}
SPL {X  -160.000, Y  +650.662, Z    +0.000, E1   -32.150, E3 +156408.900}
SPL {X  -160.000, Y  +655.372, Z    +0.000, E1   -32.145, E3 +156424.847}
SPL {X  -160.000, Y  +660.593, Z    +0.000, E1   -32.163, E3 +156442.464}
SPL {X  -160.000, Y  +665.836, Z    +0.000, E1   -32.154, E3 +156460.181}
SPL {X  -160.000, Y  +670.613, Z    +0.000, E1   -32.138, E3 +156476.391}
SPL {X  -159.954, Y  +675.336, Z    +0.000, E1   -32.135, E3 +156492.400}
SPL {X  -159.758, Y  +680.302, Z    +0.000, E1   -32.108, E3 +156509.414}
SPL {X  -159.416, Y  +685.158, Z    +0.000, E1   -32.039, E3 +156526.226}
SPL {X  -158.953, Y  +689.772, Z    +0.000, E1   -31.965, E3 +156542.325}
SPL {X  -158.363, Y  +694.328, Z    +0.000, E1   -31.871, E3 +156558.337}
SPL {X  -157.606, Y  +699.074, Z    +0.000, E1   -31.756, E3 +156575.181}
SPL {X  -156.791, Y  +703.384, Z    +0.000, E1   -31.607, E3 +156590.631}
SPL {X  -155.792, Y  +707.952, Z    +0.000, E1   -31.465, E3 +156607.077}
SPL {X  -155.149, Y  +710.598, Z    +0.000, E1   -26.183, E3 +156662.537}
ENDSPLINE

SPLINE
SPL {X  -158.679, Y  +692.020, Z    +0.000, E1   -14.212, E3 +156696.213}
SPL {X  -159.747, Y  +680.500, Z    +0.000, E1    -7.378, E3 +156704.591}
SPL {X  -160.000, Y  +671.618, Z    +0.000, E1    -1.592, E3 +156708.206}
SPL {X  -160.000, Y  +666.041, Z    +0.000, E1    +2.615, E3 +156710.172}
SPL {X  -160.000, Y  +661.396, Z    +0.000, E1    +6.484, E3 +156711.845}
SPL {X  -160.000, Y  +653.532, Z    +0.000, E1   +13.136, E3 +156715.965}
SPL {X  -160.000, Y  +631.927, Z    +0.000, E1   +26.832, E3 +156738.732}
SPL {X  -160.000, Y  +610.736, Z    +0.000, E1   +32.114, E3 +156781.401}
SPL {X  -160.000, Y  +605.907, Z    +0.000, E1   +32.114, E3 +156797.750}
SPL {X  -160.000, Y  +601.221, Z    +0.000, E1   +32.108, E3 +156813.617}
SPL {X  -160.000, Y  +596.433, Z    +0.000, E1   +32.120, E3 +156829.799}
SPL {X  -160.000, Y  +592.025, Z    +0.000, E1   +32.104, E3 +156844.724}
SPL {X  -160.000, Y  +587.734, Z    +0.000, E1   +32.110, E3 +156859.244}
SPL {X  -160.000, Y  +583.150, Z    +0.000, E1   +32.111, E3 +156874.772}
SPL {X  -160.000, Y  +579.063, Z    +0.000, E1   +32.085, E3 +156888.673}
SPL {X  -160.000, Y  +574.897, Z    +0.000, E1   +32.110, E3 +156902.724}
SPL {X  -160.000, Y  +570.471, Z    +0.000, E1   +32.093, E3 +156917.739}
SPL {X  -160.000, Y  +566.667, Z    +0.000, E1   +32.086, E3 +156930.653}
SPL {X  -160.000, Y  +562.434, Z    +0.000, E1   +32.097, E3 +156944.963}
SPL {X  -160.000, Y  +557.710, Z    +0.000, E1   +32.104, E3 +156960.946}
SPL {X  -160.000, Y  +553.479, Z    +0.000, E1   +32.081, E3 +156975.315}
SPL {X  -160.000, Y  +547.489, Z    +0.000, E1   +32.181, E3 +156995.434}
SPL {X  -160.000, Y  +541.554, Z    +0.000, E1   +32.092, E3 +157015.671}
SPL {X  -160.000, Y  +537.332, Z    +0.000, E1   +32.092, E3 +157029.968}
SPL {X  -160.000, Y  +533.113, Z    +0.000, E1   +32.090, E3 +157044.265}
SPL {X  -160.000, Y  +528.875, Z    +0.000, E1   +32.090, E3 +157058.608}
SPL {X  -160.000, Y  +524.453, Z    +0.000, E1   +32.104, E3 +157073.532}
SPL {X  -160.000, Y  +520.037, Z    +0.000, E1   +32.096, E3 +157088.474}
SPL {X  -160.000, Y  +514.030, Z    +0.000, E1   +32.182, E3 +157108.670}
SPL {X  -160.000, Y  +508.131, Z    +0.000, E1   +32.099, E3 +157128.775}
SPL {X  -160.000, Y  +504.077, Z    +0.000, E1   +32.094, E3 +157142.498}
SPL {X  -160.000, Y  +494.657, Z    +0.000, E1   +34.509, E3 +157157.361}
SPL {X  -160.000, Y  +491.565, Z    +0.000, E1   +33.823, E3 +157171.268}
SPL {X  -160.000, Y  +489.317, Z    +0.000, E1   +32.894, E3 +157184.613}
SPL {X  -160.000, Y  +486.958, Z    +0.000, E1   +31.703, E3 +157200.384}
SPL {X  -160.000, Y  +484.144, Z    +0.000, E1   +30.999, E3 +157214.807}
SPL {X  -160.000, Y  +479.156, Z    +0.000, E1   +31.035, E3 +157232.373}
SPL {X  -160.000, Y  +474.045, Z    +0.000, E1   +31.015, E3 +157250.465}
SPL {X  -160.000, Y  +468.999, Z    +0.000, E1   +31.021, E3 +157268.290}
SPL {X  -160.000, Y  +464.107, Z    +0.000, E1   +31.012, E3 +157285.590}
SPL {X  -160.000, Y  +459.262, Z    +0.000, E1   +31.016, E3 +157302.697}
SPL {X  -160.000, Y  +454.119, Z    +0.000, E1   +31.026, E3 +157320.847}
SPL {X  -160.000, Y  +448.874, Z    +0.000, E1   +31.019, E3 +157339.403}
SPL {X  -160.000, Y  +443.892, Z    +0.000, E1   +31.019, E3 +157356.991}
SPL {X  -160.000, Y  +438.782, Z    +0.000, E1   +31.022, E3 +157375.065}
SPL {X  -160.000, Y  +433.722, Z    +0.000, E1   +31.007, E3 +157393.009}
SPL {X  -160.000, Y  +428.980, Z    +0.000, E1   +31.004, E3 +157409.766}
SPL {X  -160.000, Y  +424.339, Z    +0.000, E1   +31.006, E3 +157426.140}
SPL {X  -160.000, Y  +419.231, Z    +0.000, E1   +31.030, E3 +157444.134}
SPL {X  -160.000, Y  +414.179, Z    +0.000, E1   +31.008, E3 +157462.031}
SPL {X  -160.000, Y  +409.416, Z    +0.000, E1   +31.023, E3 +157478.814}
SPL {X  -160.000, Y  +403.994, Z    +0.000, E1   +31.033, E3 +157497.970}
SPL {X  -160.000, Y  +399.052, Z    +0.000, E1   +31.010, E3 +157515.438}
SPL {X  -160.000, Y  +394.012, Z    +0.000, E1   +31.036, E3 +157533.227}
SPL {X  -159.999, Y  +388.376, Z    +0.000, E1   +31.028, E3 +157553.156}
SPL {X  -159.897, Y  +383.070, Z    +0.000, E1   +31.010, E3 +157571.994}
SPL {X  -159.656, Y  +378.313, Z    +0.000, E1   +30.961, E3 +157589.087}
SPL {X  -159.237, Y  +373.190, Z    +0.000, E1   +30.917, E3 +157607.587}
SPL {X  -158.628, Y  +367.891, Z    +0.000, E1   +30.812, E3 +157626.972}
SPL {X  -157.915, Y  +363.053, Z    +0.000, E1   +30.689, E3 +157644.839}
SPL {X  -157.216, Y  +359.084, Z    +0.000, E1   +30.550, E3 +157659.642}
SPL {X  -156.248, Y  +354.355, Z    +0.000, E1   +30.460, E3 +157677.254}
SPL {X  -155.629, Y  +351.657, Z    +0.000, E1   +25.972, E3 +157723.683}
ENDSPLINE

